(* IEC 61131-3 sources: beckhoffAutomationInterface/ST/Shark/App/Shark/FunctionBlocks, 11 files *)

(* ---- FB_ChillerManager.st ---- *)
(*
FB_ChillerManager — Controls chiller power and water valves.
Migrated from old FB_ChillerManager. Uses I_DigitalOutput from DO subsystem.
3 outputs: ChillerPower, ChuckWaterIn valve, ChuckWaterOut valve.
*)
FUNCTION_BLOCK FB_ChillerManager
VAR
    _ipChillerPower   : I_DigitalOutput;
    _ipWaterInValve   : I_DigitalOutput;
    _ipWaterOutValve  : I_DigitalOutput;
    _bInitialized     : BOOL := FALSE;
END_VAR

METHOD PUBLIC Init : BOOL
VAR_INPUT
    ipChillerPower  : I_DigitalOutput;
    ipWaterInValve  : I_DigitalOutput;
    ipWaterOutValve : I_DigitalOutput;
END_VAR
    IF ipChillerPower = 0 OR ipWaterInValve = 0 OR ipWaterOutValve = 0 THEN
        GVL_ErrorLogger.Logger.LogError(
            sSource  := 'ChillerManager.Init',
            eErrorId := E_ErrorId.ERR_GEN_NULL_POINTER,
            sContext := 'null interface pointer'
        );
        RETURN;
    END_IF
    _ipChillerPower := ipChillerPower;
    _ipWaterInValve := ipWaterInValve;
    _ipWaterOutValve := ipWaterOutValve;
    _bInitialized := TRUE;
    Init := TRUE;
END_METHOD

METHOD PUBLIC SetChillerPower
VAR_INPUT
    bOn : BOOL;
END_VAR
    _SetOutput(ipOutput := _ipChillerPower, bValue := bOn);
END_METHOD

METHOD PUBLIC SetWaterInValve
VAR_INPUT
    bOpen : BOOL;
END_VAR
    _SetOutput(ipOutput := _ipWaterInValve, bValue := bOpen);
END_METHOD

METHOD PUBLIC SetWaterOutValve
VAR_INPUT
    bOpen : BOOL;
END_VAR
    _SetOutput(ipOutput := _ipWaterOutValve, bValue := bOpen);
END_METHOD

METHOD PRIVATE _SetOutput
VAR_INPUT
    ipOutput : I_DigitalOutput;
    bValue   : BOOL;
END_VAR
    IF NOT _bInitialized THEN RETURN; END_IF
    ipOutput.SetOutput(bValue);
END_METHOD

PROPERTY PUBLIC IsChillerOn : BOOL
    GET
        IF _bInitialized AND_THEN _ipChillerPower <> 0 THEN
            IsChillerOn := _ipChillerPower.GetOutput();
        END_IF
    END_GET
END_PROPERTY

END_FUNCTION_BLOCK

(* ---- FB_ChuckVacuumSystem.st ---- *)
// Shark Chuck Vacuum System
//
// Shark hardware topology:
//   - Dedicated vacuum pump (PUMP_CHK_VAC) — toggled by this subsystem
//   - 2-way zone valves (VALV_CHK_LZ1/2/3) — open = vacuum applied
//   - Explicit vent valve (VALV_CHK_VENT) — must be closed before holding
//   - Single analog vacuum sensor (PSNS_CHK_VAC)
//
// Threshold semantics: rThreshold is in the same engineering units as the
// analog sensor; held when measurement < rThreshold, released when > rThreshold.
FUNCTION_BLOCK FB_ChuckVacuumSystem IMPLEMENTS I_ChuckVacuumSystem
VAR
    _bInitialized   : BOOL := FALSE;
    _bError         : BOOL := FALSE;

    _ipPump         : I_DigitalOutput;
    _ipValveLZ1     : I_Valve;
    _ipValveLZ2     : I_Valve;
    _ipValveLZ3     : I_Valve;
    _ipVentValve    : I_Valve;
    _ipVacuumSensor : I_Sensor;
END_VAR

VAR CONSTANT
    MAX_ZONES : INT := 3;
END_VAR

METHOD PUBLIC Init : BOOL
VAR_INPUT
    ipProvider : I_HardwareProvider;
END_VAR
    _bInitialized := FALSE;
    _bError := FALSE;

    IF ipProvider = 0 THEN
        GVL_ErrorLogger.Logger.LogError('FB_ChuckVacuumSystem', E_ErrorId.ERR_GEN_NULL_POINTER, 'Provider is null');
        RETURN;
    END_IF

    _ipPump := ipProvider.GetDigitalOutput(E_DigitalOutputIdentifier.PUMP_CHK_VAC);
    _ipValveLZ1 := ipProvider.GetValve(E_ValveIdentifier.VALV_CHK_LZ1);
    _ipValveLZ2 := ipProvider.GetValve(E_ValveIdentifier.VALV_CHK_LZ2);
    _ipValveLZ3 := ipProvider.GetValve(E_ValveIdentifier.VALV_CHK_LZ3);
    _ipVentValve := ipProvider.GetValve(E_ValveIdentifier.VALV_CHK_VENT);
    _ipVacuumSensor := ipProvider.GetPressureSensor(E_PressureSensorIdentifier.PSNS_CHK_VAC);

    IF _ipPump = 0 OR _ipValveLZ1 = 0 OR _ipVentValve = 0 OR _ipVacuumSensor = 0 THEN
        GVL_ErrorLogger.Logger.LogError('FB_ChuckVacuumSystem', E_ErrorId.ERR_GEN_NULL_POINTER, 'Required chuck vacuum hardware missing');
        RETURN;
    END_IF

    _bInitialized := TRUE;
    Init := TRUE;
END_METHOD

METHOD PUBLIC IsInitialized : BOOL
    IsInitialized := _bInitialized;
END_METHOD

METHOD PUBLIC IsError : BOOL
    IsError := _bError;
END_METHOD

METHOD PUBLIC GetMaxZoneCount : INT
    GetMaxZoneCount := MAX_ZONES;
END_METHOD

// Shark: close vent and ensure dedicated pump is on.
METHOD PUBLIC PrepareForHold : BOOL
    IF NOT _bInitialized THEN RETURN; END_IF
    _ipVentValve.Close();
    IF NOT _ipPump.GetOutput() THEN
        _ipPump.SetOutput(TRUE);
    END_IF
    PrepareForHold := TRUE;
END_METHOD

// Shark: open vent to atmosphere. Caller closes zones separately.
METHOD PUBLIC BeginRelease : BOOL
    IF NOT _bInitialized THEN RETURN; END_IF
    _ipVentValve.Open();
    BeginRelease := TRUE;
END_METHOD

// Shark: turn off dedicated chuck vacuum pump.
METHOD PUBLIC FinishRelease : BOOL
    IF NOT _bInitialized THEN RETURN; END_IF
    _ipPump.SetOutput(FALSE);
    FinishRelease := TRUE;
END_METHOD

METHOD PUBLIC OpenZone : BOOL
VAR_INPUT
    nZone : INT;
END_VAR
    OpenZone := _SetZoneState(nZone := nZone, bOpen := TRUE);
END_METHOD

METHOD PUBLIC CloseZone : BOOL
VAR_INPUT
    nZone : INT;
END_VAR
    CloseZone := _SetZoneState(nZone := nZone, bOpen := FALSE);
END_METHOD

// Analog sensor: vacuum held when pressure < threshold.
// nActiveZoneCount is ignored — single sensor measures shared vacuum manifold.
METHOD PUBLIC IsVacuumHeld : BOOL
VAR_INPUT
    nActiveZoneCount : INT;
    rThreshold       : LREAL;
END_VAR
    IF NOT _bInitialized THEN RETURN; END_IF
    IsVacuumHeld := (_ipVacuumSensor.GetMeasurement() < rThreshold);
END_METHOD

// Analog sensor: vacuum released when pressure > threshold.
METHOD PUBLIC IsVacuumReleased : BOOL
VAR_INPUT
    rThreshold : LREAL;
END_VAR
    IF NOT _bInitialized THEN RETURN; END_IF
    IsVacuumReleased := (_ipVacuumSensor.GetMeasurement() > rThreshold);
END_METHOD

METHOD PUBLIC Reset : BOOL
    _bError := FALSE;
    IF _ipValveLZ1 <> 0 AND_THEN _ipValveLZ1.IsError() THEN _ipValveLZ1.Reset(); END_IF
    IF _ipValveLZ2 <> 0 AND_THEN _ipValveLZ2.IsError() THEN _ipValveLZ2.Reset(); END_IF
    IF _ipValveLZ3 <> 0 AND_THEN _ipValveLZ3.IsError() THEN _ipValveLZ3.Reset(); END_IF
    IF _ipVentValve <> 0 AND_THEN _ipVentValve.IsError() THEN _ipVentValve.Reset(); END_IF
    Reset := TRUE;
END_METHOD

METHOD PRIVATE _SetZoneState : BOOL
VAR_INPUT
    nZone : INT;
    bOpen : BOOL;
END_VAR
    IF NOT _bInitialized THEN RETURN; END_IF

    CASE nZone OF
        1:
            IF _ipValveLZ1 = 0 THEN RETURN; END_IF
            IF bOpen THEN _ipValveLZ1.Open(); ELSE _ipValveLZ1.Close(); END_IF
        2:
            IF _ipValveLZ2 = 0 THEN RETURN; END_IF
            IF bOpen THEN _ipValveLZ2.Open(); ELSE _ipValveLZ2.Close(); END_IF
        3:
            IF _ipValveLZ3 = 0 THEN RETURN; END_IF
            IF bOpen THEN _ipValveLZ3.Open(); ELSE _ipValveLZ3.Close(); END_IF
        ELSE
            RETURN;
    END_CASE

    _SetZoneState := TRUE;
END_METHOD

END_FUNCTION_BLOCK

(* ---- FB_CommandReceiver.st ---- *)
(*
FB_CommandReceiver — Receives JSON commands from ADS byte stream and dispatches
to hardware provider, spectrometer, and sequence engine.

ADS Pattern:
  DALP Manager (.NET) writes JSON as raw bytes into AdsStream[0..4095].
  This FB polls every scan: if non-zero → parse JSON → dispatch → clear buffer.

Debug:
  Each command has a corresponding stDbgXxx struct and bDbgTrigXxx BOOL.
  Set struct fields and trigger from TwinCAT online to execute any command
  through the same code path as the Pilot.

Handles all command types from E_Command:
  Subsystem:    SetValve, SetMFCFlowRate, SetPressureController, SetHeaterZone,
                SetSwitch, ErrorAcknowledge
  Sequence:     SetTemperatureGradients, CancelProcess, StartBubblerFlow,
                StopBubblerFlow, StartPurge, HoldReleaseSample,
                StartSpotDeposition, StartBubblerLeakTest
  Spectrometer: SetSpectrometerData, SetSpectrometerDark

Requires Tc3_JsonXml library for FB_JsonDomParser + FB_JsonReadWriteDataType.
*)
FUNCTION_BLOCK FB_CommandReceiver
VAR
    AdsStream              : ARRAY[0..4095] OF BYTE;
    ZeroArray              : ARRAY[0..4095] OF BYTE;
    sCommand               : STRING(4096);
    sLastCommandParsed     : STRING(4096);
    SuccessCommandCount    : UDINT := 0;
    ErrorCommandCount      : UDINT := 0;

    fbJson                 : FB_JsonDomParser;
    jsonDoc                : Tc3_JsonXml.PVOID;
    jsonProp               : SJsonValue;
    fbJsonDataType         : FB_JsonReadWriteDataType;

    _nCommand              : DINT;
    _nCommandIndex         : DINT;

    _ipHardware            : I_HardwareProvider;
    _ipSpectrometer        : I_Spectrometer;
    _refOrchestrator       : REFERENCE TO FB_SequenceOrchestrator;
    _rTempDisableThreshold : REAL := 0.0;   // degC if any zone's setpoint is below this, disable all commands that could heat
    _bInitialized          : BOOL := FALSE;

    // Debug: set struct fields + trigger from TwinCAT online to test any command
    // Subsystem
    stDbgSetValve              : ST_CmdSetValve;
    bDbgTrigSetValve           : BOOL;
    stDbgSetFlowRate           : ST_CmdSetFlowRate;
    bDbgTrigSetFlowRate        : BOOL;
    stDbgSetPressure           : ST_CmdSetPressure;
    bDbgTrigSetPressure        : BOOL;
    stDbgSetHeatZone           : ST_CmdSetHeatZone;
    bDbgTrigSetHeatZone        : BOOL;
    stDbgSetSwitch             : ST_CmdSetSwitch;
    bDbgTrigSetSwitch          : BOOL;
    bDbgTrigErrorAck           : BOOL;
    // Sequence
    stDbgTempGradient          : ST_CmdSetTemperatureGradient;
    bDbgTrigTempGradient       : BOOL;
    bDbgTrigCancelProcess      : BOOL;
    stDbgBubblerFlow           : ST_CmdStartBubblerFlow;
    bDbgTrigBubblerFlow        : BOOL;
    stDbgStopBubblerFlow       : ST_CmdStopBubblerFlow;
    bDbgTrigStopBubblerFlow    : BOOL;
    stDbgPurge                 : ST_CmdPurge;
    bDbgTrigPurge              : BOOL;
    stDbgChuckZone             : ST_CmdSetChuckZone;
    bDbgTrigChuckZone          : BOOL;
    stDbgSpotDeposition        : ST_CmdSpotDeposition;
    bDbgTrigSpotDeposition     : BOOL;
    stDbgLeakTest              : ST_CmdBubblerLeakTest;
    bDbgTrigLeakTest           : BOOL;
    // Spectrometer
    stDbgSpectrometerData      : ST_DeviceSettings;
    bDbgTrigSpectrometerData   : BOOL;
    bDbgTrigSpectrometerDark   : BOOL;
END_VAR
VAR_OUTPUT
    nLastCommandIndex      : DINT;
END_VAR
VAR CONSTANT
    JSON_KEY_COMMAND             : STRING := 'command';
    JSON_KEY_INDEX               : STRING := 'index';
    JSON_KEY_PARAMETERS          : STRING := 'parameters';
    JSON_PARAM_BUFFER_SIZE       : UDINT  := 2048;
    // Minimum flow rate above which the inert gas inlet valve is opened.
    // At or below this threshold the valve is closed.
    INERT_FLOW_VALVE_THRESHOLD   : REAL   := 0.001;
END_VAR

    IF NOT _bInitialized THEN
        RETURN;
    END_IF

    IF MEMCMP(ADR(AdsStream), ADR(ZeroArray), SIZEOF(AdsStream)) <> 0 THEN
        sCommand := _ByteArrToString(ADR(AdsStream), SIZEOF(AdsStream));
        IF _ParseAndDispatch() THEN
            SuccessCommandCount := SuccessCommandCount + 1;
        ELSE
            ErrorCommandCount := ErrorCommandCount + 1;
        END_IF
        MEMSET(ADR(AdsStream), 0, SIZEOF(AdsStream));
        sLastCommandParsed := sCommand;
    END_IF

    // Debug triggers (set params + trigger from TwinCAT online)
    _ProcessDebugTriggers();

METHOD PUBLIC Init : BOOL
VAR_INPUT
    ipHardware     : I_HardwareProvider;
    ipSpectrometer : I_Spectrometer;
    rTempDisableThreshold : REAL;
    refOrchestrator : REFERENCE TO FB_SequenceOrchestrator;
END_VAR
    IF ipHardware = 0 OR ipSpectrometer = 0 THEN
        GVL_ErrorLogger.Logger.LogError(
            sSource  := 'CommandReceiver.Init',
            eErrorId := E_ErrorId.ERR_GEN_NULL_POINTER,
            sContext := 'invalid interface'
        );
        RETURN;
    END_IF
    IF NOT __ISVALIDREF(refOrchestrator) THEN
        GVL_ErrorLogger.Logger.LogError(
            sSource  := 'CommandReceiver.Init',
            eErrorId := E_ErrorId.ERR_GEN_NULL_POINTER,
            sContext := 'invalid orchestrator reference'
        );
        RETURN;
    END_IF
    _ipHardware            := ipHardware;
    _ipSpectrometer        := ipSpectrometer;
    _rTempDisableThreshold := rTempDisableThreshold;
    _refOrchestrator       REF= refOrchestrator;
    _bInitialized          := TRUE;
    Init := TRUE;
END_METHOD

METHOD PRIVATE _ParseAndDispatch : BOOL
VAR
    nError         : INT := 0;
    stSetValve     : ST_CmdSetValve;
    stSetFlowRate  : ST_CmdSetFlowRate;
    stSetPressure  : ST_CmdSetPressure;
    stSetHeatZone  : ST_CmdSetHeatZone;
    stSetHeatChannel : ST_CmdSetHeatChannel;
    stSetSwitch    : ST_CmdSetSwitch;
    stTempGrad     : ST_CmdSetTemperatureGradient;
    stBubblerFlow  : ST_CmdStartBubblerFlow;
    stStopBubbler  : ST_CmdStopBubblerFlow;
    stPurge        : ST_CmdPurge;
    stChuckZone    : ST_CmdSetChuckZone;
    stSpotDep      : ST_CmdSpotDeposition;
    stLeakTest     : ST_CmdBubblerLeakTest;
    stSpecData     : ST_DeviceSettings;
    eCmd           : E_Command;
END_VAR
    jsonDoc := fbJson.ParseDocument(sCommand);

    jsonProp := fbJson.FindMember(jsonDoc, JSON_KEY_COMMAND);
    IF jsonProp <> 0 THEN
        _nCommand := fbJson.GetInt(jsonProp);
    ELSE
        GVL_ErrorLogger.Logger.LogError(
            sSource   := 'CommandReceiver',
            eErrorId  := E_ErrorId.ERR_GEN_INVALID_PARAM,
            sContext  := 'missing command field in JSON',
            eSeverity := E_TcEventSeverity.Warning
        );
        _ParseAndDispatch := FALSE;
        RETURN;
    END_IF

    jsonProp := fbJson.FindMember(jsonDoc, JSON_KEY_INDEX);
    IF jsonProp <> 0 THEN
        _nCommandIndex := fbJson.GetInt(jsonProp);
    END_IF

    eCmd := DINT_TO_INT(_nCommand);
    CASE eCmd OF
        E_Command.SetValve:
            IF _ParseJsonParams('ST_CmdSetValve', SIZEOF(stSetValve), ADR(stSetValve)) THEN
                nError := _CmdSetValve(stCmd := stSetValve);
            ELSE nError := -1; END_IF
        E_Command.SetMFCFlowRate:
            IF _ParseJsonParams('ST_CmdSetFlowRate', SIZEOF(stSetFlowRate), ADR(stSetFlowRate)) THEN
                nError := _CmdSetMFCFlowRate(stCmd := stSetFlowRate);
            ELSE nError := -1; END_IF
        E_Command.SetPressureController:
            IF _ParseJsonParams('ST_CmdSetPressure', SIZEOF(stSetPressure), ADR(stSetPressure)) THEN
                nError := _CmdSetPressure(stCmd := stSetPressure);
            ELSE nError := -1; END_IF
        E_Command.SetHeaterZone:
            IF _ParseJsonParams('ST_CmdSetHeatZone', SIZEOF(stSetHeatZone), ADR(stSetHeatZone)) THEN
                nError := _CmdSetHeatZone(stCmd := stSetHeatZone);
            ELSE nError := -1; END_IF
        E_Command.SetHeaterChannel:
            IF _ParseJsonParams('ST_CmdSetHeatChannel', SIZEOF(stSetHeatChannel), ADR(stSetHeatChannel)) THEN
                nError := _CmdSetHeatChannel(stCmd := stSetHeatChannel);
            ELSE nError := -1; END_IF
        E_Command.SetSwitch:
            IF _ParseJsonParams('ST_CmdSetSwitch', SIZEOF(stSetSwitch), ADR(stSetSwitch)) THEN
                nError := _CmdSetSwitch(stCmd := stSetSwitch);
            ELSE nError := -1; END_IF
        E_Command.ErrorAcknowledge:
            nError := _CmdErrorAcknowledge();
        E_Command.SetTemperatureGradients:
            IF _ParseJsonParams('ST_CmdSetTemperatureGradient', SIZEOF(stTempGrad), ADR(stTempGrad)) THEN
                nError := _CmdSetTemperatureGradient(stCmd := stTempGrad);
            ELSE nError := -1; END_IF
        E_Command.CancelProcess:
            nError := _CmdCancelProcess();
        E_Command.StartBubblerFlow:
            IF _ParseJsonParams('ST_CmdStartBubblerFlow', SIZEOF(stBubblerFlow), ADR(stBubblerFlow)) THEN
                nError := _CmdStartBubblerFlow(stCmd := stBubblerFlow);
            ELSE nError := -1; END_IF
        E_Command.StopBubblerFlow:
            IF _ParseJsonParams('ST_CmdStopBubblerFlow', SIZEOF(stStopBubbler), ADR(stStopBubbler)) THEN
                nError := _CmdStopBubblerFlow(stCmd := stStopBubbler);
            ELSE nError := -1; END_IF
        E_Command.StartPurge:
            IF _ParseJsonParams('ST_CmdPurge', SIZEOF(stPurge), ADR(stPurge)) THEN
                nError := _CmdStartPurge(stCmd := stPurge);
            ELSE nError := -1; END_IF
        E_Command.HoldReleaseSample:
            IF _ParseJsonParams('ST_CmdSetChuckZone', SIZEOF(stChuckZone), ADR(stChuckZone)) THEN
                nError := _CmdHoldReleaseSample(stCmd := stChuckZone);
            ELSE nError := -1; END_IF
        E_Command.StartSpotDeposition:
            IF _ParseJsonParams('ST_CmdSpotDeposition', SIZEOF(stSpotDep), ADR(stSpotDep)) THEN
                nError := _CmdStartSpotDeposition(stCmd := stSpotDep);
            ELSE nError := -1; END_IF
        E_Command.StartBubblerLeakTest:
            IF _ParseJsonParams('ST_CmdBubblerLeakTest', SIZEOF(stLeakTest), ADR(stLeakTest)) THEN
                nError := _CmdStartBubblerLeakTest(stCmd := stLeakTest);
            ELSE nError := -1; END_IF
        E_Command.SetSpectrometerData:
            IF _ParseJsonParams('ST_DeviceSettings', SIZEOF(stSpecData), ADR(stSpecData)) THEN
                nError := _CmdSetSpectrometerData(stSettings := stSpecData);
            ELSE nError := -1; END_IF
        E_Command.SetSpectrometerDark:
            nError := _CmdSetSpectrometerDark();
    ELSE
        GVL_ErrorLogger.Logger.LogError(
            sSource   := 'CommandReceiver',
            eErrorId  := E_ErrorId.ERR_GEN_INVALID_PARAM,
            sContext  := CONCAT('unknown command ', CONCAT(TO_STRING(eCmd), CONCAT(' (', CONCAT(DINT_TO_STRING(_nCommand), ')')))),
            eSeverity := E_TcEventSeverity.Warning
        );
        _ParseAndDispatch := FALSE;
        RETURN;
    END_CASE

    IF nError = 0 THEN
        nLastCommandIndex := _nCommandIndex;
        _ParseAndDispatch := TRUE;
    ELSE
        GVL_ErrorLogger.Logger.LogError(
            sSource   := 'CommandReceiver',
            eErrorId  := E_ErrorId.ERR_GEN_INTERNAL,
            sContext  := CONCAT('command failed ', CONCAT(TO_STRING(eCmd), CONCAT(' (', CONCAT(DINT_TO_STRING(_nCommand), ')')))),
            eSeverity := E_TcEventSeverity.Warning
        );
        _ParseAndDispatch := FALSE;
    END_IF
END_METHOD

METHOD PRIVATE _ParseJsonParams : BOOL
VAR_INPUT
    sTypeName : STRING;
    nSize     : UDINT;
    pDest     : PVOID;
END_VAR
VAR
    sParamJson : STRING(JSON_PARAM_BUFFER_SIZE);
    nLen       : UDINT;
END_VAR
    jsonProp := fbJson.FindMember(jsonDoc, JSON_KEY_PARAMETERS);
    IF jsonProp = 0 THEN
        // No 'parameters' wrapper — fall back to using the full JSON directly
        sParamJson := sCommand;
    ELSE
        nLen := fbJson.GetJsonLength(jsonProp);
        fbJson.CopyJson(jsonProp, sParamJson, nLen);
    END_IF

    IF NOT fbJsonDataType.SetSymbolFromJson(sParamJson, sTypeName, nSize, pDest) THEN
        GVL_ErrorLogger.Logger.LogError(
            sSource   := 'CommandReceiver',
            eErrorId  := E_ErrorId.ERR_GEN_INVALID_PARAM,
            sContext  := CONCAT('failed to parse ', sTypeName),
            eSeverity := E_TcEventSeverity.Warning
        );
        _ParseJsonParams := FALSE;
        RETURN;
    END_IF
    _ParseJsonParams := TRUE;
END_METHOD

// =============================================================================
// COMMAND HANDLERS — Pure execution, no JSON parsing
// =============================================================================

METHOD PRIVATE _CmdSetValve : INT
VAR_INPUT
    stCmd : ST_CmdSetValve;
END_VAR
VAR
    ipValve : I_Valve;
    eValve  : E_ValveIdentifier;
END_VAR
    eValve := stCmd.valveId;
    GVL_ErrorLogger.Logger.LogInfo(
        sSource  := 'CommandReceiver',
        sContext := CONCAT('SetValve(', CONCAT(DINT_TO_STRING(_nCommand), CONCAT('): ', CONCAT(TO_STRING(eValve), CONCAT('(', CONCAT(INT_TO_STRING(stCmd.valveId), CONCAT(') enabled=', BOOL_TO_STRING(stCmd.enabled))))))))
    );
    ipValve := _ipHardware.GetValve(stCmd.valveId);
    IF ipValve <> 0 THEN
        IF stCmd.enabled THEN
            ipValve.Open();
        ELSE
            ipValve.Close();
        END_IF
    ELSE
        _CmdSetValve := -1;
    END_IF
END_METHOD

METHOD PRIVATE _CmdSetMFCFlowRate : INT
VAR_INPUT
    stCmd : ST_CmdSetFlowRate;
END_VAR
VAR
    ipController : I_Controller;
    ipInertValve : I_Valve;
    eMFC         : E_MFCIdentifier;
END_VAR
    eMFC := stCmd.mfcId;
    GVL_ErrorLogger.Logger.LogInfo(
        sSource  := 'CommandReceiver',
        sContext := CONCAT('SetMFCFlowRate(', CONCAT(DINT_TO_STRING(_nCommand), CONCAT('): ', CONCAT(TO_STRING(eMFC), CONCAT('(', CONCAT(INT_TO_STRING(stCmd.mfcId), CONCAT(') flowRate=', REAL_TO_STRING(stCmd.flowRate))))))))
    );
    ipController := _ipHardware.GetFlowController(stCmd.mfcId);
    IF ipController <> 0 THEN
        ipController.SetSetpoint(stCmd.flowRate);
        // When the inert MFC (MFCT_IG_01) is commanded, also control its inlet valve.
        IF eMFC = E_MFCIdentifier.MFCT_IG_01 THEN
            ipInertValve := _ipHardware.GetInertGasValve();
            IF ipInertValve <> 0 THEN
                IF stCmd.flowRate > INERT_FLOW_VALVE_THRESHOLD THEN
                    ipInertValve.Open();
                ELSE
                    ipInertValve.Close();
                END_IF
            END_IF
        END_IF
    ELSE
        _CmdSetMFCFlowRate := -1;
    END_IF
END_METHOD

METHOD PRIVATE _CmdSetPressure : INT
VAR_INPUT
    stCmd : ST_CmdSetPressure;
END_VAR
VAR
    ipController : I_Controller;
    ePressure    : E_PressureController;
END_VAR
    ePressure := stCmd.psctrlId;
    GVL_ErrorLogger.Logger.LogInfo(
        sSource  := 'CommandReceiver',
        sContext := CONCAT('SetPressureController(', CONCAT(DINT_TO_STRING(_nCommand), CONCAT('): ', CONCAT(TO_STRING(ePressure), CONCAT('(', CONCAT(INT_TO_STRING(stCmd.psctrlId), CONCAT(') pressure=', REAL_TO_STRING(stCmd.pressure))))))))
    );
    ipController := _ipHardware.GetPressureControllerById(stCmd.psctrlId);
    IF ipController <> 0 THEN
        ipController.SetSetpoint(stCmd.pressure);
    ELSE
        _CmdSetPressure := -1;
    END_IF
END_METHOD

METHOD PRIVATE _CmdSetHeatZone : INT
VAR_INPUT
    stCmd : ST_CmdSetHeatZone;
END_VAR
VAR
    ipController : I_Controller;
    eLegacyZone  : E_HeatZones;   // per-channel id sent by the DALP/Pilot client (1..15)
    eZone        : E_HeatZone;    // internal controllable zone id (1..13)
END_VAR
    // The legacy DALP/Pilot client addresses heater CHANNELS via E_HeatZones
    // (1..15), but SetHeaterZone operates on ZONES via E_HeatZone (1..13).
    // Reject any id that is not a defined E_HeatZones member, then translate.
    eLegacyZone := stCmd.zoneId;
    IF NOT _LegacyChannelToZone(eLegacy := eLegacyZone, eZone => eZone) THEN
        GVL_ErrorLogger.Logger.LogError(
            sSource   := 'CommandReceiver.SetHeatZone',
            eErrorId  := E_ErrorId.ERR_GEN_INVALID_PARAM,
            sContext  := CONCAT('invalid zoneId ', INT_TO_STRING(stCmd.zoneId)),
            eSeverity := E_TcEventSeverity.Warning
        );
        _CmdSetHeatZone := -1;
        RETURN;
    END_IF

    GVL_ErrorLogger.Logger.LogInfo(
        sSource  := 'CommandReceiver',
        sContext := CONCAT('SetHeatZone(', CONCAT(DINT_TO_STRING(_nCommand), CONCAT('): ', CONCAT(TO_STRING(eLegacyZone), CONCAT(' -> ', CONCAT(TO_STRING(eZone), CONCAT(' temp=', REAL_TO_STRING(stCmd.temp))))))))
    );

    ipController := _ipHardware.GetTemperatureController(eZone);
    IF ipController <> 0 THEN
        IF stCmd.temp > _rTempDisableThreshold THEN
            ipController.SetSetpoint(stCmd.temp);
            ipController.Enable(TRUE);
        ELSE
            ipController.Enable(FALSE);
        END_IF
    ELSE
        _CmdSetHeatZone := -1;
    END_IF
END_METHOD

(* Translate the legacy per-CHANNEL id (E_HeatZones, 1..15 — what the DALP/Pilot
   client sends) into the internal controllable ZONE id (E_HeatZone, 1..13).
   The 11 single-channel zones map 1:1. The two 2-channel zones each have two
   legacy channel ids that both resolve to the single owning zone:
       HETR_EXH_01 / HETR_EXH_02 -> HETR_EXH
       HETR_CHK_01 / HETR_CHK_02 -> HETR_CHK
   Commanding either channel id therefore enables the whole zone (FB_HeatZone
   fans Enable() out to every channel it owns).
   Returns TRUE and sets eZone on success; returns FALSE (leaving eZone
   untouched) for any value that is not a defined E_HeatZones member, so the
   caller can fail the command instead of acting on a wrong zone. *)
METHOD PRIVATE _LegacyChannelToZone : BOOL
VAR_INPUT
    eLegacy : E_HeatZones;
END_VAR
VAR_OUTPUT
    eZone : E_HeatZone;
END_VAR
    _LegacyChannelToZone := TRUE;
    CASE eLegacy OF
        E_HeatZones.HETR_HEAD_01 : eZone := E_HeatZone.HETR_HEAD;
        E_HeatZones.HETR_A_STR_01: eZone := E_HeatZone.HETR_A_STR;
        E_HeatZones.HETR_A_CMB_01: eZone := E_HeatZone.HETR_A_CMB;
        E_HeatZones.HETR_A_B1_01 : eZone := E_HeatZone.HETR_A_B1;
        E_HeatZones.HETR_A_B2_01 : eZone := E_HeatZone.HETR_A_B2;
        E_HeatZones.HETR_A_B3_01 : eZone := E_HeatZone.HETR_A_B3;
        E_HeatZones.HETR_B_STR_01: eZone := E_HeatZone.HETR_B_STR;
        E_HeatZones.HETR_B_CMB_01: eZone := E_HeatZone.HETR_B_CMB;
        E_HeatZones.HETR_B_B1_01 : eZone := E_HeatZone.HETR_B_B1;
        E_HeatZones.HETR_B_B2_01 : eZone := E_HeatZone.HETR_B_B2;
        E_HeatZones.HETR_B_B3_01 : eZone := E_HeatZone.HETR_B_B3;
        E_HeatZones.HETR_EXH_01,
        E_HeatZones.HETR_EXH_02  : eZone := E_HeatZone.HETR_EXH;
        E_HeatZones.HETR_CHK_01,
        E_HeatZones.HETR_CHK_02  : eZone := E_HeatZone.HETR_CHK;
    ELSE
        // Unknown id — not a defined E_HeatZones member. Fail; do not guess.
        _LegacyChannelToZone := FALSE;
    END_CASE
END_METHOD

METHOD PRIVATE _CmdSetHeatChannel : INT
VAR_INPUT
    stCmd : ST_CmdSetHeatChannel;
END_VAR
VAR
    ipController : I_Controller;
    eChannel     : E_HeatChannel;
END_VAR
    eChannel := stCmd.channelId;
    GVL_ErrorLogger.Logger.LogInfo(
        sSource  := 'CommandReceiver',
        sContext := CONCAT('SetHeatChannel(', CONCAT(DINT_TO_STRING(_nCommand), CONCAT('): ', CONCAT(TO_STRING(eChannel), CONCAT('(', CONCAT(INT_TO_STRING(stCmd.channelId), CONCAT(') temp=', REAL_TO_STRING(stCmd.temp))))))))
    );
    ipController := _ipHardware.GetTemperatureChannel(stCmd.channelId);
    IF ipController <> 0 THEN
        IF stCmd.temp > _rTempDisableThreshold THEN
            ipController.SetSetpoint(stCmd.temp);
            ipController.Enable(TRUE);
        ELSE
            ipController.Enable(FALSE);
        END_IF
    ELSE
        _CmdSetHeatChannel := -1;
    END_IF
END_METHOD

METHOD PRIVATE _CmdSetSwitch : INT
VAR_INPUT
    stCmd : ST_CmdSetSwitch;
END_VAR
VAR
    ipOutput : I_DigitalOutput;
    eDIO     : E_DIOIdentifier;
    eOutput  : E_DigitalOutputIdentifier;
END_VAR
    // switchId is sent by DALP Manager as an E_DIOIdentifier value (telemetry index 1..25).
    // Translate to E_DigitalOutputIdentifier before addressing the hardware.
    eDIO := stCmd.switchId;
    GVL_ErrorLogger.Logger.LogInfo(
        sSource  := 'CommandReceiver',
        sContext := CONCAT('SetSwitch(', CONCAT(DINT_TO_STRING(_nCommand), CONCAT('): ', CONCAT(TO_STRING(eDIO), CONCAT('(', CONCAT(INT_TO_STRING(stCmd.switchId), CONCAT(') enabled=', BOOL_TO_STRING(stCmd.enabled))))))))
    );

    CASE eDIO OF
        E_DIOIdentifier.LGHT_CMR_SIDE : eOutput := E_DigitalOutputIdentifier.LGHT_CMR_SIDE;
        E_DIOIdentifier.LGHT_CMR_TOP  : eOutput := E_DigitalOutputIdentifier.LGHT_CMR_TOP;
        E_DIOIdentifier.CHIL_PWR      : eOutput := E_DigitalOutputIdentifier.CHIL_PWR;
        // LGHT_SGN_RED, LGHT_SGN_YEL, LGHT_SGN_GRN are owned by FB_SignalLightController — not manually settable.
        E_DIOIdentifier.LOCK_DOOR_FL  : eOutput := E_DigitalOutputIdentifier.LOCK_DOOR_FL;
        E_DIOIdentifier.LOCK_DOOR_FR  : eOutput := E_DigitalOutputIdentifier.LOCK_DOOR_FR;
        E_DIOIdentifier.PUMP_CHK_VAC  : eOutput := E_DigitalOutputIdentifier.PUMP_CHK_VAC;
        E_DIOIdentifier.VALV_CHK_LZ1  : eOutput := E_DigitalOutputIdentifier.VALV_CHK_LZ1;
        E_DIOIdentifier.VALV_CHK_LZ2  : eOutput := E_DigitalOutputIdentifier.VALV_CHK_LZ2;
        E_DIOIdentifier.VALV_CHK_LZ3  : eOutput := E_DigitalOutputIdentifier.VALV_CHK_LZ3;
        E_DIOIdentifier.VALV_CHK_VENT : eOutput := E_DigitalOutputIdentifier.VALV_CHK_VENT;
    ELSE
        // DIO indices 9-17 are digital inputs (PRXS_DOOR_*) — not writable outputs.
        // DIO indices 24-25 are safety inputs (SAFE_STO_ON, SAFE_OVERRIDE) — not writable.
        GVL_ErrorLogger.Logger.LogError(
            sSource   := 'CommandReceiver.SetSwitch',
            eErrorId  := E_ErrorId.ERR_GEN_INVALID_PARAM,
            sContext  := CONCAT('DIO index ', CONCAT(TO_STRING(eDIO), ' is not a writable digital output')),
            eSeverity := E_TcEventSeverity.Warning
        );
        _CmdSetSwitch := -1;
        RETURN;
    END_CASE

    ipOutput := _ipHardware.GetDigitalOutput(eOutput);
    IF ipOutput <> 0 THEN
        ipOutput.SetOutput(stCmd.enabled);
    ELSE
        _CmdSetSwitch := -1;
    END_IF
END_METHOD

METHOD PRIVATE _CmdSetTemperatureGradient : INT
VAR_INPUT
    stCmd : ST_CmdSetTemperatureGradient;
END_VAR
    GVL_ErrorLogger.Logger.LogInfo(
        sSource  := 'CommandReceiver',
        sContext := CONCAT('SetTemperatureGradients: mode=', CONCAT(INT_TO_STRING(stCmd.enableMode), CONCAT(' head=', REAL_TO_STRING(stCmd.headTemp))))
    );
    IF NOT _refOrchestrator.StartHeating(stParams := stCmd) THEN
        _CmdSetTemperatureGradient := -1;
    END_IF
END_METHOD

METHOD PRIVATE _CmdErrorAcknowledge : INT
    GVL_System.bGlobalEmergencyStop := FALSE;
    _refOrchestrator.ErrorAcknowledge();
    GVL_ErrorLogger.Logger.LogInfo(
        sSource  := 'CommandReceiver',
        sContext := 'ErrorAcknowledge received'
    );
END_METHOD

METHOD PRIVATE _CmdCancelProcess : INT
    GVL_ErrorLogger.Logger.LogInfo(
        sSource  := 'CommandReceiver',
        sContext := 'CancelProcess'
    );
    IF NOT _refOrchestrator.SystemStop() THEN
        _CmdCancelProcess := -1;
    END_IF
END_METHOD

METHOD PRIVATE _CmdStartBubblerFlow : INT
VAR_INPUT
    stCmd : ST_CmdStartBubblerFlow;
END_VAR
VAR
    eSide : E_GasSide;
END_VAR
    eSide := stCmd.side;
    GVL_ErrorLogger.Logger.LogInfo(
        sSource  := 'CommandReceiver',
        sContext := CONCAT('StartBubblerFlow(', CONCAT(DINT_TO_STRING(_nCommand), CONCAT('): side=', CONCAT(TO_STRING(eSide), CONCAT('(', CONCAT(INT_TO_STRING(stCmd.side), CONCAT(') flow=', CONCAT(REAL_TO_STRING(stCmd.flowRate), CONCAT(' bubbler=', INT_TO_STRING(stCmd.bubblerIndex))))))))))
    );
    IF NOT _refOrchestrator.StartBubblerFlow(stParams := stCmd) THEN
        _CmdStartBubblerFlow := -1;
    END_IF
END_METHOD

METHOD PRIVATE _CmdStopBubblerFlow : INT
VAR_INPUT
    stCmd : ST_CmdStopBubblerFlow;
END_VAR
VAR
    eSide : E_GasSide;
END_VAR
    eSide := stCmd.side;
    GVL_ErrorLogger.Logger.LogInfo(
        sSource  := 'CommandReceiver',
        sContext := CONCAT('StopBubblerFlow(', CONCAT(DINT_TO_STRING(_nCommand), CONCAT('): side=', CONCAT(TO_STRING(eSide), CONCAT('(', CONCAT(INT_TO_STRING(stCmd.side), ')'))))))
    );
    IF NOT _refOrchestrator.StopBubblerFlow(stParams := stCmd) THEN
        _CmdStopBubblerFlow := -1;
    END_IF
END_METHOD

METHOD PRIVATE _CmdStartPurge : INT
VAR_INPUT
    stCmd : ST_CmdPurge;
END_VAR
VAR
    eMode : E_PurgeMode;
    eSide : E_GasSide;
END_VAR
    eMode := stCmd.mode;
    eSide := stCmd.side;
    GVL_ErrorLogger.Logger.LogInfo(
        sSource  := 'CommandReceiver',
        sContext := CONCAT('StartPurge(', CONCAT(DINT_TO_STRING(_nCommand), CONCAT('): ', CONCAT(TO_STRING(eMode), CONCAT('(', CONCAT(INT_TO_STRING(stCmd.mode), CONCAT(') side=', CONCAT(TO_STRING(eSide), CONCAT('(', CONCAT(INT_TO_STRING(stCmd.side), CONCAT(') bubbler=', INT_TO_STRING(stCmd.bubbler))))))))))))
    );
    IF NOT _refOrchestrator.StartPurge(stParams := stCmd) THEN
        _CmdStartPurge := -1;
    END_IF
END_METHOD

METHOD PRIVATE _CmdHoldReleaseSample : INT
VAR_INPUT
    stCmd     : ST_CmdSetChuckZone;
END_VAR
VAR
    iZone     : INT;
    stHold    : ST_ChuckVacuumHold;
    stRelease : ST_ChuckVacuumRelease;
END_VAR
    GVL_ErrorLogger.Logger.LogInfo(
        sSource  := 'CommandReceiver',
        sContext := CONCAT('HoldReleaseSample: hold=', CONCAT(BOOL_TO_STRING(stCmd.holdSample), CONCAT(' waferSize=', INT_TO_STRING(stCmd.size))))
    );
    IF stCmd.size < GVL_ChuckVacuumSystem.CHUCK_ZONE_SMALL_MAX THEN
        iZone := 1;
    ELSIF stCmd.size < GVL_ChuckVacuumSystem.CHUCK_ZONE_MEDIUM_MAX THEN
        iZone := 2;
    ELSE
        iZone := 3;
    END_IF

    IF stCmd.holdSample THEN
        stHold.iSelectZone := iZone;
        stHold.fLockPressureThreshold := stCmd.fPressureThreshold;
        stHold.tPressureTimeout := DINT_TO_TIME(stCmd.tPressureTimeout);
        IF NOT _refOrchestrator.StartChuckVacuumHold(stParams := stHold) THEN
            _CmdHoldReleaseSample := -1;
        END_IF
    ELSE
        stRelease.fReleasePressureThreshold := stCmd.fPressureThreshold;
        stRelease.tPressureTimeout := DINT_TO_TIME(stCmd.tPressureTimeout);
        IF NOT _refOrchestrator.StartChuckVacuumRelease(stParams := stRelease) THEN
            _CmdHoldReleaseSample := -1;
        END_IF
    END_IF
END_METHOD

METHOD PRIVATE _CmdStartSpotDeposition : INT
VAR_INPUT
    stCmd : ST_CmdSpotDeposition;
END_VAR
    GVL_ErrorLogger.Logger.LogInfo(
        sSource  := 'CommandReceiver',
        sContext := CONCAT('StartSpotDeposition: cycles=', CONCAT(DINT_TO_STRING(stCmd.nDepositionCycles), CONCAT(' precFlow=', REAL_TO_STRING(stCmd.fPrecursorFlowRate))))
    );
    IF NOT _refOrchestrator.StartSpotDeposition(stParams := stCmd) THEN
        _CmdStartSpotDeposition := -1;
    END_IF
END_METHOD

METHOD PRIVATE _CmdStartBubblerLeakTest : INT
VAR_INPUT
    stCmd : ST_CmdBubblerLeakTest;
END_VAR
VAR
    eSide : E_GasSide;
END_VAR
    eSide := stCmd.side;
    GVL_ErrorLogger.Logger.LogInfo(
        sSource  := 'CommandReceiver',
        sContext := CONCAT('StartBubblerLeakTest(', CONCAT(DINT_TO_STRING(_nCommand), CONCAT('): side=', CONCAT(TO_STRING(eSide), CONCAT('(', CONCAT(INT_TO_STRING(stCmd.side), CONCAT(') bubbler=', DINT_TO_STRING(stCmd.bubblerIndex))))))))
    );
    IF NOT _refOrchestrator.StartBubblerLeakTest(stParams := stCmd) THEN
        _CmdStartBubblerLeakTest := -1;
    END_IF
END_METHOD

METHOD PRIVATE _CmdSetSpectrometerData : INT
VAR_INPUT
    stSettings : ST_DeviceSettings;
END_VAR
    GVL_ErrorLogger.Logger.LogInfo(
        sSource  := 'CommandReceiver',
        sContext := CONCAT('SetSpectrometerData: scanRate=', CONCAT(UDINT_TO_STRING(stSettings.ScanRate), CONCAT(' avg=', UDINT_TO_STRING(stSettings.SpectrumAverage))))
    );
    _ipSpectrometer.SetFrequency(stSettings.ScanRate);
    _ipSpectrometer.SetLightIntensity(
        TargetLight := stSettings.LightTargetPercentage,
        AutoAdjust  := stSettings.IntensityAutoAdjust
    );
    _ipSpectrometer.SetAverageSample(stSettings.SpectrumAverage);
    _ipSpectrometer.SetSpectrumLimits(
        nStartRatio  := stSettings.SpectrumStart,
        nStopRatio   := stSettings.SpectrumStop,
        nTotalPixels := INT_TO_UDINT(GVL_Spectrometer.SPECTROMETER_PIXEL_COUNT)
    );
    _ipSpectrometer.SetQualityTreshold(stSettings.QualityThresholdPercentage);
END_METHOD

METHOD PRIVATE _CmdSetSpectrometerDark : INT
    GVL_ErrorLogger.Logger.LogInfo(
        sSource  := 'CommandReceiver',
        sContext := 'SetSpectrometerDark'
    );
    _ipSpectrometer.CalibrateDark(bExecute := TRUE);
END_METHOD

// =============================================================================
// DEBUG TRIGGERS — TwinCAT online: set struct fields, set trigger BOOL
// =============================================================================

METHOD PRIVATE _ProcessDebugTriggers
    // Subsystem
    IF bDbgTrigSetValve THEN
        bDbgTrigSetValve := FALSE;
        _CmdSetValve(stCmd := stDbgSetValve);
    END_IF
    IF bDbgTrigSetFlowRate THEN
        bDbgTrigSetFlowRate := FALSE;
        _CmdSetMFCFlowRate(stCmd := stDbgSetFlowRate);
    END_IF
    IF bDbgTrigSetPressure THEN
        bDbgTrigSetPressure := FALSE;
        _CmdSetPressure(stCmd := stDbgSetPressure);
    END_IF
    IF bDbgTrigSetHeatZone THEN
        bDbgTrigSetHeatZone := FALSE;
        _CmdSetHeatZone(stCmd := stDbgSetHeatZone);
    END_IF
    IF bDbgTrigSetSwitch THEN
        bDbgTrigSetSwitch := FALSE;
        _CmdSetSwitch(stCmd := stDbgSetSwitch);
    END_IF
    IF bDbgTrigErrorAck THEN
        bDbgTrigErrorAck := FALSE;
        _CmdErrorAcknowledge();
    END_IF

    // Sequence
    IF bDbgTrigTempGradient THEN
        bDbgTrigTempGradient := FALSE;
        _CmdSetTemperatureGradient(stCmd := stDbgTempGradient);
    END_IF
    IF bDbgTrigCancelProcess THEN
        bDbgTrigCancelProcess := FALSE;
        _CmdCancelProcess();
    END_IF
    IF bDbgTrigBubblerFlow THEN
        bDbgTrigBubblerFlow := FALSE;
        _CmdStartBubblerFlow(stCmd := stDbgBubblerFlow);
    END_IF
    IF bDbgTrigStopBubblerFlow THEN
        bDbgTrigStopBubblerFlow := FALSE;
        _CmdStopBubblerFlow(stCmd := stDbgStopBubblerFlow);
    END_IF
    IF bDbgTrigPurge THEN
        bDbgTrigPurge := FALSE;
        _CmdStartPurge(stCmd := stDbgPurge);
    END_IF
    IF bDbgTrigChuckZone THEN
        bDbgTrigChuckZone := FALSE;
        _CmdHoldReleaseSample(stCmd := stDbgChuckZone);
    END_IF
    IF bDbgTrigSpotDeposition THEN
        bDbgTrigSpotDeposition := FALSE;
        _CmdStartSpotDeposition(stCmd := stDbgSpotDeposition);
    END_IF
    IF bDbgTrigLeakTest THEN
        bDbgTrigLeakTest := FALSE;
        _CmdStartBubblerLeakTest(stCmd := stDbgLeakTest);
    END_IF

    // Spectrometer
    IF bDbgTrigSpectrometerData THEN
        bDbgTrigSpectrometerData := FALSE;
        _CmdSetSpectrometerData(stSettings := stDbgSpectrometerData);
    END_IF
    IF bDbgTrigSpectrometerDark THEN
        bDbgTrigSpectrometerDark := FALSE;
        _CmdSetSpectrometerDark();
    END_IF
END_METHOD

METHOD PRIVATE _ByteArrToString : STRING(4096)
VAR_INPUT
    pbyBuf : POINTER TO BYTE;
    diLen  : DINT;
END_VAR
VAR
    sResult  : STRING(4096) := '';
    nCopyLen : DINT;
END_VAR
    nCopyLen := MIN(diLen, 4095);
    MEMCPY(ADR(sResult), pbyBuf, TO_UDINT(nCopyLen));
    _ByteArrToString := sResult;
END_METHOD

END_FUNCTION_BLOCK

(* ---- FB_DALP.st ---- *)
(*
FB_DALP — Legacy client compatibility wrapper.

Exposes the exact ADS symbol contract the old C# DALP Manager expects:
  * MAIN.fbDALP.stTelemetry  (ST_Atlant3d_Telemetry, alias of ST_MachineTelemetry)
  * MAIN.fbDALP.AdsStream    (ARRAY[0..4095] OF BYTE, command write path)

This FB does not own any subsystem logic. It is a thin pass-through:
  1. Each scan, copy the new publisher's stTelemetry into our own
     stTelemetry (struct types alias each other, so the assignment is
     byte-for-byte equivalent).
  2. Overwrite the HETR_ array per-CHANNEL (not per-zone) so the legacy
     client's E_HeatZones iteration (15 entries) gets the right data.
  3. Forward any bytes the client wrote into AdsStream to the receiver's
     buffer, then clear the local buffer.

DELETE THIS FOLDER ONCE THE CLIENT IS UPDATED. See README.md.
*)
FUNCTION_BLOCK FB_DALP
VAR
    stTelemetry       : ST_Atlant3d_Telemetry;
    AdsStream         : ARRAY[0..4095] OF BYTE;
    _ZeroArray        : ARRAY[0..4095] OF BYTE;

    _refPublisher     : REFERENCE TO FB_TelemetryPublisher;
    _refReceiver      : REFERENCE TO FB_CommandReceiver;
    _refTempSub       : REFERENCE TO FB_TemperatureSubsystem;

    _bInitialized     : BOOL := FALSE;
END_VAR

    IF NOT _bInitialized THEN
        RETURN;
    END_IF

    // 1. Mirror the new publisher's full telemetry (identical struct shape via alias)
    stTelemetry := _refPublisher.stTelemetry;

    // 2. Re-fill HETR_ per-CHANNEL for the legacy client (15 entries on Shark)
    _UpdateHeatersPerChannel();

    // 3. Forward any client-written command bytes to the receiver
    IF MEMCMP(ADR(AdsStream), ADR(_ZeroArray), SIZEOF(AdsStream)) <> 0 THEN
        MEMCPY(
            destAddr := ADR(_refReceiver.AdsStream),
            srcAddr  := ADR(AdsStream),
            n        := SIZEOF(AdsStream)
        );
        MEMSET(ADR(AdsStream), 0, SIZEOF(AdsStream));
    END_IF

METHOD PUBLIC Init : BOOL
VAR_INPUT
    refPublisher : REFERENCE TO FB_TelemetryPublisher;
    refReceiver  : REFERENCE TO FB_CommandReceiver;
    refTempSub   : REFERENCE TO FB_TemperatureSubsystem;
END_VAR
    IF NOT __ISVALIDREF(refPublisher) THEN RETURN; END_IF
    IF NOT __ISVALIDREF(refReceiver)  THEN RETURN; END_IF
    IF NOT __ISVALIDREF(refTempSub)   THEN RETURN; END_IF

    _refPublisher REF= refPublisher;
    _refReceiver  REF= refReceiver;
    _refTempSub   REF= refTempSub;
    _bInitialized := TRUE;
    Init := TRUE;
END_METHOD

(* Per-CHANNEL heater telemetry for the legacy client.
   Iterates every (zone, channel) pair and writes HETR_[globalIdx]. *)
{attribute 'estimated-stack-usage' := '500'}
METHOD PRIVATE _UpdateHeatersPerChannel
VAR
    iZone       : INT;
    c           : INT;
    nCount      : INT;
    nGlobalIdx  : INT;
    ipChannel   : I_Controller;
    stCtrl      : ST_ControllerStatus;
END_VAR
    FOR iZone := 1 TO GVL_TemperatureZones.CONTROLLABLE_ZONE_MAX DO
        nCount := GVL_TemperatureZoneConfig.ZONE_CONFIG[iZone].nChannelCount;
        FOR c := 1 TO nCount DO
            nGlobalIdx := _refTempSub.GetChannelGlobalIndex(eZone := iZone, nChannelIdx := c);
            IF nGlobalIdx < 1 THEN CONTINUE; END_IF

            ipChannel := _refTempSub.GetChannel(eZone := iZone, nChannelIdx := c);
            IF ipChannel = 0 THEN CONTINUE; END_IF

            stCtrl := ipChannel.GetStatus();
            stTelemetry.HETR_[nGlobalIdx].Enable             := stCtrl.bEnabled;
            stTelemetry.HETR_[nGlobalIdx].TempAvg            := TO_REAL(stCtrl.rMeasuredValue);
            stTelemetry.HETR_[nGlobalIdx].SP                 := TO_REAL(stCtrl.rSetpoint);
            stTelemetry.HETR_[nGlobalIdx].TemperatureReached := stCtrl.bAtSetpoint;
            stTelemetry.HETR_[nGlobalIdx].Status             := SEL(
                stCtrl.stError.eErrorId = E_ErrorId.NO_ERROR, INT#1, INT#0);
        END_FOR
    END_FOR
END_METHOD

END_FUNCTION_BLOCK

(* ---- FB_DoorsManager.st ---- *)
(*
FB_DoorsManager — Shark-specific door wiring. Implements I_DoorSystem (Facade).

Facade pattern: presents the I_DoorSystem surface to sequence and safety code;
hides the lock/sensor graph and all Shark identifier knowledge from callers.

Layout: 9 proximity sensors, 2 door locks.
  Lock 1 FL (Front Left)  → sensors PRXS_DOOR_LT, PRXS_DOOR_LM
  Lock 2 FR (Front Right) → sensors PRXS_DOOR_RT, PRXS_DOOR_RM
  Remaining sensors (LB, RB, BML, BMR, BMB) are standalone monitoring only.

Sensor index assumption: E_DigitalInputIdentifier door enum values are dense
and align 1:1 with _afbSensors[1..SENSOR_COUNT]. If the enum is renumbered
this mapping must be revisited.
*)
FUNCTION_BLOCK FB_DoorsManager IMPLEMENTS I_DoorSystem
VAR
    _afbSensors   : ARRAY[1..GVL_DoorSystem.DOOR_SENSOR_COUNT] OF FB_DoorSensor;
    _afbLocks     : ARRAY[1..GVL_DoorSystem.DOOR_LOCK_COUNT] OF FB_DoorLock;
    _bInitialized : BOOL := FALSE;
END_VAR

METHOD PUBLIC Init : BOOL
VAR_INPUT
    ipDISub : I_DigitalInputSubsystem;
    ipDOSub : I_DigitalOutputSubsystem;
END_VAR
VAR
    i : INT;
END_VAR
    IF ipDISub = 0 OR ipDOSub = 0 THEN
        GVL_ErrorLogger.Logger.LogError(
            sSource  := 'DoorsManager.Init',
            eErrorId := E_ErrorId.ERR_GEN_NULL_POINTER,
            sContext := 'invalid subsystem interface pointer'
        );
        RETURN;
    END_IF

    // Initialise all 9 standalone monitoring sensors.
    // Relies on dense enum alignment: sensor identifier i maps to _afbSensors[i].
    FOR i := 1 TO GVL_DoorSystem.DOOR_SENSOR_COUNT DO
        _afbSensors[i].Init(ipInput := ipDISub.GetInputByIndex(nInput := i));
    END_FOR

    // Lock 1 — Front Left
    _afbLocks[1].Init(
        ipOutput := ipDOSub.GetOutputByIndex(nOutput := E_DigitalOutputIdentifier.LOCK_DOOR_FL)
    );
    _afbLocks[1].AddSensor(ipInput := ipDISub.GetInputByIndex(nInput := E_DigitalInputIdentifier.PRXS_DOOR_LT));
    _afbLocks[1].AddSensor(ipInput := ipDISub.GetInputByIndex(nInput := E_DigitalInputIdentifier.PRXS_DOOR_LM));

    // Lock 2 — Front Right
    _afbLocks[2].Init(
        ipOutput := ipDOSub.GetOutputByIndex(nOutput := E_DigitalOutputIdentifier.LOCK_DOOR_FR)
    );
    _afbLocks[2].AddSensor(ipInput := ipDISub.GetInputByIndex(nInput := E_DigitalInputIdentifier.PRXS_DOOR_RT));
    _afbLocks[2].AddSensor(ipInput := ipDISub.GetInputByIndex(nInput := E_DigitalInputIdentifier.PRXS_DOOR_RM));

    _bInitialized := TRUE;
    Init := TRUE;
END_METHOD

METHOD PUBLIC IsDoorClosed : BOOL
VAR_INPUT
    nSensorIndex : INT;
END_VAR
    IF nSensorIndex >= 1 AND nSensorIndex <= GVL_DoorSystem.DOOR_SENSOR_COUNT THEN
        IsDoorClosed := _afbSensors[nSensorIndex].IsClosed;
    END_IF
END_METHOD

METHOD PUBLIC IsLockActivated : BOOL
VAR_INPUT
    nLockIndex : INT;
END_VAR
    IF nLockIndex >= 1 AND nLockIndex <= GVL_DoorSystem.DOOR_LOCK_COUNT THEN
        IsLockActivated := _afbLocks[nLockIndex].IsLocked;
    END_IF
END_METHOD

METHOD PUBLIC LockDoor
VAR_INPUT
    nLockIndex : INT;
END_VAR
    IF nLockIndex >= 1 AND nLockIndex <= GVL_DoorSystem.DOOR_LOCK_COUNT THEN
        _afbLocks[nLockIndex].Lock();
    END_IF
END_METHOD

METHOD PUBLIC UnlockDoor
VAR_INPUT
    nLockIndex : INT;
END_VAR
    IF nLockIndex >= 1 AND nLockIndex <= GVL_DoorSystem.DOOR_LOCK_COUNT THEN
        _afbLocks[nLockIndex].Unlock();
    END_IF
END_METHOD

METHOD PUBLIC AreAllDoorsClosed : BOOL
VAR
    i : INT;
END_VAR
    AreAllDoorsClosed := TRUE;
    FOR i := 1 TO GVL_DoorSystem.DOOR_SENSOR_COUNT DO
        IF NOT _afbSensors[i].IsClosed THEN
            AreAllDoorsClosed := FALSE;
            RETURN;
        END_IF
    END_FOR
END_METHOD

END_FUNCTION_BLOCK

(* ---- FB_ExhaustController.st ---- *)
(*
FB_ExhaustController — Exhaust pump controller.

Keeps the exhaust pump energised at all times and optionally verifies
operation via an isolation valve and pressure sensor.

Configuration variants (set at Init time):
  A. Valve before sensor (bIsoValveBeforeSensor=TRUE, Shark):
       PUMP_ON → OPENING_VALVE → WAIT_PRESSURE → READY
  B. Sensor before valve, or no valve (bIsoValveBeforeSensor=FALSE):
       PUMP_ON → WAIT_PRESSURE → READY   (valve not managed here)
  C. Sensor only, no valve:
       PUMP_ON → WAIT_PRESSURE → READY
  D. Neither:
       PUMP_ON → READY

Pump output is re-driven every scan cycle — it cannot be silenced by
Halt() calls or any other external writer.
*)
FUNCTION_BLOCK FB_ExhaustController
VAR CONSTANT
    PRESSURE_THRESHOLD : LREAL := 0.4;   // bar — minimum to confirm pump health
    ISO_VALVE_OPEN_TIMEOUT  : TIME  := T#10S; // maximum wait for IsOpen() to return TRUE
    PRESSURE_BUILD_TIMEOUT  : TIME  := T#60S; // maximum wait for pressure to reach threshold
END_VAR
VAR
    _ipExhaustPump          : I_DigitalOutput;
    _ipIsoValve             : I_Valve;
    _ipPressureSensor       : I_Sensor;
    _bIsoValveBeforeSensor : BOOL;
    _eState                : E_ExhaustState := E_ExhaustState.INIT;
    _tonIsoValveOpen       : TON;
    _tonPressureBuild      : TON;
    _bInitialized           : BOOL := FALSE;
END_VAR

    IF NOT _bInitialized THEN
        RETURN;
    END_IF

    // Re-drive every scan — prevents any external SetOutput(FALSE) from lasting more than one cycle
    _ipExhaustPump.SetOutput(TRUE);

    CASE _eState OF

        E_ExhaustState.INIT:
            _eState := E_ExhaustState.PUMP_ON;

        E_ExhaustState.PUMP_ON:
            IF _ipIsoValve <> 0 AND_THEN _bIsoValveBeforeSensor THEN
                _eState := E_ExhaustState.OPENING_VALVE;
            ELSIF _ipPressureSensor <> 0 THEN
                _eState := E_ExhaustState.WAIT_PRESSURE;
            ELSE
                _eState := E_ExhaustState.READY;
            END_IF

        E_ExhaustState.OPENING_VALVE:
            _ipIsoValve.Open();
            _tonIsoValveOpen(IN := TRUE, PT := ISO_VALVE_OPEN_TIMEOUT);
            IF _ipIsoValve.IsOpen() THEN
                _tonIsoValveOpen(IN := FALSE);
                IF _ipPressureSensor <> 0 THEN
                    _eState := E_ExhaustState.WAIT_PRESSURE;
                ELSE
                    _eState := E_ExhaustState.READY;
                END_IF
            ELSIF _tonIsoValveOpen.Q THEN
                GVL_ErrorLogger.Logger.LogError(
                    sSource  := 'ExhaustController',
                    eErrorId := E_ErrorId.ERR_VALVE_FEEDBACK_TIMEOUT,
                    sContext := 'iso valve did not open within timeout',
                    fCurrentValue  := TO_REAL(TIME_TO_DWORD(_tonIsoValveOpen.ET)) / 1000.0,
                    fExpectedValue := TO_REAL(TIME_TO_DWORD(ISO_VALVE_OPEN_TIMEOUT)) / 1000.0,
                    sUnits := 's'
                );
                _eState := E_ExhaustState.ERROR;
            END_IF

        E_ExhaustState.WAIT_PRESSURE:
            _tonPressureBuild(IN := TRUE, PT := PRESSURE_BUILD_TIMEOUT);
            IF _ipPressureSensor.GetMeasurement() >= PRESSURE_THRESHOLD THEN
                _tonPressureBuild(IN := FALSE);
                _eState := E_ExhaustState.READY;
            ELSIF _tonPressureBuild.Q THEN
                GVL_ErrorLogger.Logger.LogError(
                    sSource  := 'ExhaustController',
                    eErrorId := E_ErrorId.ERR_GEN_TIMEOUT,
                    sContext := 'pressure threshold not reached',
                    fCurrentValue  := TO_REAL(_ipPressureSensor.GetMeasurement()),
                    fExpectedValue := TO_REAL(PRESSURE_THRESHOLD),
                    sUnits := 'bar'
                );
                _eState := E_ExhaustState.ERROR;
            END_IF

        E_ExhaustState.READY:
            ; // Pump always on — nothing to monitor

        E_ExhaustState.ERROR:
            ; // Stays here until Reset()

    END_CASE

METHOD PUBLIC Init : BOOL
VAR_INPUT
    ipExhaustPump          : I_DigitalOutput;
    ipIsoValve             : I_Valve  := 0;    // Optional — 0 if machine has no iso valve
    ipPressureSensor       : I_Sensor := 0;    // Optional — 0 if machine has no pressure sensor
    bIsoValveBeforeSensor  : BOOL     := FALSE; // TRUE = iso valve sits between pump and sensor (Shark);
                                                 // pressure is not meaningful until valve is open
END_VAR
    IF ipExhaustPump = 0 THEN
        GVL_ErrorLogger.Logger.LogError(
            sSource  := 'ExhaustController.Init',
            eErrorId := E_ErrorId.ERR_GEN_NULL_POINTER,
            sContext := 'null pump interface'
        );
        RETURN;
    END_IF
    _ipExhaustPump          := ipExhaustPump;
    _ipIsoValve             := ipIsoValve;
    _ipPressureSensor       := ipPressureSensor;
    _bIsoValveBeforeSensor  := bIsoValveBeforeSensor;
    _bInitialized           := TRUE;
    _eState                 := E_ExhaustState.INIT;
    Init := TRUE;
END_METHOD

METHOD PUBLIC Reset
    IF _bInitialized THEN
        _tonIsoValveOpen(IN := FALSE);
        _tonPressureBuild(IN := FALSE);
        IF _ipIsoValve <> 0 THEN
            _ipIsoValve.Close();
        END_IF
        _eState := E_ExhaustState.INIT;
    END_IF
END_METHOD

PROPERTY PUBLIC IsReady : BOOL
    GET
        IsReady := _eState = E_ExhaustState.READY;
    END_GET
END_PROPERTY

PROPERTY PUBLIC State : E_ExhaustState
    GET
        State := _eState;
    END_GET
END_PROPERTY

END_FUNCTION_BLOCK

(* ---- FB_HardwareProvider.st ---- *)
(* Hardware provider for Shark System (Dual-sided gas, Modbus pressure).
   Delegates Init and index-based subsystem access to FB_HardwareProviderBase.

   Shark-specific differences from PRO:
   - Per-side mix valves (VALV_A_MIX, VALV_B_MIX) instead of shared VALV_AB_MIX
   - Separate CM and HM vacuum isolation (DST_EXH vs CMB_EXH) instead of shared exhaust
   - Modbus pressure controllers via E_PressureController
    - 3 bubblers per side (no B-side gas-only lines)
    - No inert MFC side mapping (accessed via generic GetValve) *)
FUNCTION_BLOCK FB_HardwareProvider EXTENDS FB_HardwareProviderBase IMPLEMENTS I_HardwareProvider
VAR
    _nMaxBubblers : ARRAY[1..2] OF DINT := [3, 3];  // index matches E_GasSide: A_SIDE=1 → 3, B_SIDE=2 → 3
    _fbChuckVacuum         : FB_ChuckVacuumSystem;
    _bChuckVacuumInitTried : BOOL := FALSE;
END_VAR

// =============================================================================
// GENERIC GETTERS — thin wrappers delegating to base index-based helpers
// =============================================================================

METHOD GetValve : I_Valve
VAR_INPUT
    nIndex : INT;
END_VAR
    GetValve := SUPER^.GetValveByIndex(nIndex);
END_METHOD

METHOD GetDigitalOutput : I_DigitalOutput
VAR_INPUT
    nIndex : INT;
END_VAR
    GetDigitalOutput := SUPER^.GetOutputByIndex(nIndex);
END_METHOD

METHOD GetDigitalInput : I_DigitalInput
VAR_INPUT
    nIndex : INT;
END_VAR
    GetDigitalInput := SUPER^.GetInputByIndex(nIndex);
END_METHOD

METHOD GetPressureSensor : I_Sensor
VAR_INPUT
    nIndex : INT;
END_VAR
    GetPressureSensor := SUPER^.GetSensorByIndex(nIndex);
END_METHOD

METHOD GetFlowController : I_Controller
VAR_INPUT
    nIndex : INT;
END_VAR
    GetFlowController := SUPER^.GetFlowControllerByIndex(nIndex);
END_METHOD

METHOD GetPressureControllerById : I_Controller
VAR_INPUT
    nIndex : INT;
END_VAR
    GetPressureControllerById := SUPER^.GetPressureControllerByIndex(nIndex);
END_METHOD

METHOD GetTemperatureController : I_Controller
VAR_INPUT
    nIndex : INT;
END_VAR
    GetTemperatureController := SUPER^.GetTemperatureControllerByIndex(nIndex);
END_METHOD

METHOD GetTemperatureChannel : I_Controller
VAR_INPUT
    nGlobalIdx : INT;
END_VAR
    GetTemperatureChannel := SUPER^.GetTemperatureChannelByGlobalIndex(nGlobalIdx);
END_METHOD

// =============================================================================
// VALVE GETTERS - Side-abstracted
// =============================================================================

// Shark: One MFC valve per side (no extra gas lines)
METHOD GetGasIsoValve : I_Valve
VAR_INPUT
    eSide : E_GasSide;
    nBubblerIndex : DINT;
END_VAR
    IF eSide = E_GasSide.A_SIDE THEN
        GetGasIsoValve := GetValve(E_ValveIdentifier.VALV_A_MFC01);
    ELSE
        GetGasIsoValve := GetValve(E_ValveIdentifier.VALV_B_MFC01);
    END_IF
END_METHOD

// CM (Distributor) bubbler inlet valves
METHOD GetCMBubblerValve : I_Valve
VAR_INPUT
    eSide : E_GasSide;
    nBubblerIndex : DINT;
END_VAR
    nBubblerIndex := LIMIT(1, nBubblerIndex, 3);

    IF eSide = E_GasSide.A_SIDE THEN
        CASE nBubblerIndex OF
            1: GetCMBubblerValve := GetValve(E_ValveIdentifier.VALV_A_DST_B1);
            2: GetCMBubblerValve := GetValve(E_ValveIdentifier.VALV_A_DST_B2);
            3: GetCMBubblerValve := GetValve(E_ValveIdentifier.VALV_A_DST_B3);
        END_CASE
    ELSE
        CASE nBubblerIndex OF
            1: GetCMBubblerValve := GetValve(E_ValveIdentifier.VALV_B_DST_B1);
            2: GetCMBubblerValve := GetValve(E_ValveIdentifier.VALV_B_DST_B2);
            3: GetCMBubblerValve := GetValve(E_ValveIdentifier.VALV_B_DST_B3);
        END_CASE
    END_IF
END_METHOD

// HM (Combiner) bubbler outlet valves
METHOD GetHMBubblerValve : I_Valve
VAR_INPUT
    eSide : E_GasSide;
    nBubblerIndex : DINT;
END_VAR
    nBubblerIndex := LIMIT(1, nBubblerIndex, 3);

    IF eSide = E_GasSide.A_SIDE THEN
        CASE nBubblerIndex OF
            1: GetHMBubblerValve := GetValve(E_ValveIdentifier.VALV_A_CMB_B1);
            2: GetHMBubblerValve := GetValve(E_ValveIdentifier.VALV_A_CMB_B2);
            3: GetHMBubblerValve := GetValve(E_ValveIdentifier.VALV_A_CMB_B3);
        END_CASE
    ELSE
        CASE nBubblerIndex OF
            1: GetHMBubblerValve := GetValve(E_ValveIdentifier.VALV_B_CMB_B1);
            2: GetHMBubblerValve := GetValve(E_ValveIdentifier.VALV_B_CMB_B2);
            3: GetHMBubblerValve := GetValve(E_ValveIdentifier.VALV_B_CMB_B3);
        END_CASE
    END_IF
END_METHOD

METHOD GetCMPurgeValve : I_Valve
VAR_INPUT
    eSide : E_GasSide;
END_VAR
    IF eSide = E_GasSide.A_SIDE THEN
        GetCMPurgeValve := GetValve(E_ValveIdentifier.VALV_A_DST_PRG);
    ELSE
        GetCMPurgeValve := GetValve(E_ValveIdentifier.VALV_B_DST_PRG);
    END_IF
END_METHOD

METHOD GetHMPurgeValve : I_Valve
VAR_INPUT
    eSide : E_GasSide;
END_VAR
    IF eSide = E_GasSide.A_SIDE THEN
        GetHMPurgeValve := GetValve(E_ValveIdentifier.VALV_A_CMB_PRG);
    ELSE
        GetHMPurgeValve := GetValve(E_ValveIdentifier.VALV_B_CMB_PRG);
    END_IF
END_METHOD

// Shark: Separate CM and HM vacuum isolation (Distributor Exhaust vs Combiner Exhaust)
METHOD GetCMVacuumIsoValve : I_Valve
VAR_INPUT
    eSide : E_GasSide;
END_VAR
    IF eSide = E_GasSide.A_SIDE THEN
        GetCMVacuumIsoValve := GetValve(E_ValveIdentifier.VALV_A_DST_EXH);
    ELSE
        GetCMVacuumIsoValve := GetValve(E_ValveIdentifier.VALV_B_DST_EXH);
    END_IF
END_METHOD

METHOD GetHMVacuumIsoValve : I_Valve
VAR_INPUT
    eSide : E_GasSide;
END_VAR
    IF eSide = E_GasSide.A_SIDE THEN
        GetHMVacuumIsoValve := GetValve(E_ValveIdentifier.VALV_A_CMB_EXH);
    ELSE
        GetHMVacuumIsoValve := GetValve(E_ValveIdentifier.VALV_B_CMB_EXH);
    END_IF
END_METHOD

METHOD GetNozzleIsoValve : I_Valve
VAR_INPUT
    eSide : E_GasSide;
END_VAR
    IF eSide = E_GasSide.A_SIDE THEN
        GetNozzleIsoValve := GetValve(E_ValveIdentifier.VALV_A_STR);
    ELSE
        GetNozzleIsoValve := GetValve(E_ValveIdentifier.VALV_B_STR);
    END_IF
END_METHOD

// =============================================================================
// VALVE GETTERS - Common
// =============================================================================

// Shark has per-side mix valves (VALV_A_MIX, VALV_B_MIX), no shared mix valve.
// Returns 0 — use GetValve(E_ValveIdentifier.VALV_A_MIX) for direct access.
METHOD GetMixValve : I_Valve
    GetMixValve := 0;
END_METHOD

METHOD GetExhaustVacuumIsoValve : I_Valve
    GetExhaustVacuumIsoValve := GetValve(E_ValveIdentifier.VALV_EX_PUMP);
END_METHOD

// =============================================================================
// DIGITAL OUTPUT GETTERS
// =============================================================================

METHOD GetExhaustPump : I_DigitalOutput
    GetExhaustPump := GetDigitalOutput(E_DigitalOutputIdentifier.PUMP_AB_EXH);
END_METHOD

// =============================================================================
// SENSOR GETTERS - Side-abstracted
// =============================================================================

// CM (Distributor) pressure sensors
METHOD GetCMPressureSensor : I_Sensor
VAR_INPUT
    eSide : E_GasSide;
END_VAR
    IF eSide = E_GasSide.A_SIDE THEN
        GetCMPressureSensor := GetPressureSensor(E_PressureSensorIdentifier.PSNS_A_DST);
    ELSE
        GetCMPressureSensor := GetPressureSensor(E_PressureSensorIdentifier.PSNS_B_DST);
    END_IF
END_METHOD

// HM (Combiner/Hot Manifold) — Bronkhorst controller as sensor via __QUERYINTERFACE
METHOD GetHMPressureSensor : I_Sensor
VAR_INPUT
    eSide : E_GasSide;
END_VAR
    IF eSide = E_GasSide.A_SIDE THEN
        GetHMPressureSensor := SUPER^.GetPressureControllerAsSensor(E_PressureController.A_Side);
    ELSE
        GetHMPressureSensor := SUPER^.GetPressureControllerAsSensor(E_PressureController.B_Side);
    END_IF
END_METHOD

METHOD GetMFCFlowSensor : I_Sensor
VAR_INPUT
    eSide : E_GasSide;
END_VAR
    IF eSide = E_GasSide.A_SIDE THEN
        GetMFCFlowSensor := SUPER^.GetFlowControllerAsSensor(E_MFCIdentifier.MFCT_A_01);
    ELSE
        GetMFCFlowSensor := SUPER^.GetFlowControllerAsSensor(E_MFCIdentifier.MFCT_B_01);
    END_IF
END_METHOD

// =============================================================================
// SENSOR GETTERS - Common
// =============================================================================

METHOD GetExhaustPressureSensor : I_Sensor
    GetExhaustPressureSensor := GetPressureSensor(E_PressureSensorIdentifier.PSNS_AB_EXH);
END_METHOD

// =============================================================================
// CONTROLLER GETTERS - Side-abstracted
// =============================================================================

METHOD GetMFCController : I_Controller
VAR_INPUT
    eSide : E_GasSide;
END_VAR
    IF eSide = E_GasSide.A_SIDE THEN
        GetMFCController := SUPER^.GetFlowControllerByIndex(E_MFCIdentifier.MFCT_A_01);
    ELSE
        GetMFCController := SUPER^.GetFlowControllerByIndex(E_MFCIdentifier.MFCT_B_01);
    END_IF
END_METHOD

// Shark: Modbus Bronkhorst pressure controllers (E_PressureController)
METHOD GetPressureController : I_Controller
VAR_INPUT
    eSide : E_GasSide;
END_VAR
    IF eSide = E_GasSide.A_SIDE THEN
        GetPressureController := SUPER^.GetPressureControllerByIndex(E_PressureController.A_Side);
    ELSE
        GetPressureController := SUPER^.GetPressureControllerByIndex(E_PressureController.B_Side);
    END_IF
END_METHOD

// Inert Gas MFC Controller (Shark-only, used by SpotDeposition)
METHOD GetInertMFCController : I_Controller
    GetInertMFCController := SUPER^.GetFlowControllerByIndex(E_MFCIdentifier.MFCT_IG_01);
END_METHOD

// Inert Gas Valve (used by SpotDeposition)
METHOD GetInertGasValve : I_Valve
    GetInertGasValve := GetValve(E_ValveIdentifier.VALV_IG_MFC01);
END_METHOD

// Chuck Vacuum Subsystem — lazy-initialized on first request.
METHOD GetChuckVacuumSystem : I_ChuckVacuumSystem
    IF NOT _bChuckVacuumInitTried THEN
        _bChuckVacuumInitTried := TRUE;
        _fbChuckVacuum.Init(ipProvider := THIS^);
    END_IF
    GetChuckVacuumSystem := _fbChuckVacuum;
END_METHOD

// =============================================================================
// TEMPERATURE CONTROLLER GETTERS - Side-abstracted
// =============================================================================

METHOD GetHMTemperatureController : I_Controller
VAR_INPUT
    eSide : E_GasSide;
END_VAR
    IF eSide = E_GasSide.A_SIDE THEN
        GetHMTemperatureController := SUPER^.GetTemperatureControllerByIndex(E_HeatZone.HETR_A_CMB);
    ELSE
        GetHMTemperatureController := SUPER^.GetTemperatureControllerByIndex(E_HeatZone.HETR_B_CMB);
    END_IF
END_METHOD

METHOD GetUmbilicalTemperatureController : I_Controller
VAR_INPUT
    eSide : E_GasSide;
END_VAR
    IF eSide = E_GasSide.A_SIDE THEN
        GetUmbilicalTemperatureController := SUPER^.GetTemperatureControllerByIndex(E_HeatZone.HETR_A_STR);
    ELSE
        GetUmbilicalTemperatureController := SUPER^.GetTemperatureControllerByIndex(E_HeatZone.HETR_B_STR);
    END_IF
END_METHOD

METHOD GetBubblerTemperatureController : I_Controller
VAR_INPUT
    eSide : E_GasSide;
    nBubblerIndex : DINT;
END_VAR
    nBubblerIndex := LIMIT(1, nBubblerIndex, 3);

    IF eSide = E_GasSide.A_SIDE THEN
        CASE nBubblerIndex OF
            1: GetBubblerTemperatureController := SUPER^.GetTemperatureControllerByIndex(E_HeatZone.HETR_A_B1);
            2: GetBubblerTemperatureController := SUPER^.GetTemperatureControllerByIndex(E_HeatZone.HETR_A_B2);
            3: GetBubblerTemperatureController := SUPER^.GetTemperatureControllerByIndex(E_HeatZone.HETR_A_B3);
        END_CASE
    ELSE
        CASE nBubblerIndex OF
            1: GetBubblerTemperatureController := SUPER^.GetTemperatureControllerByIndex(E_HeatZone.HETR_B_B1);
            2: GetBubblerTemperatureController := SUPER^.GetTemperatureControllerByIndex(E_HeatZone.HETR_B_B2);
            3: GetBubblerTemperatureController := SUPER^.GetTemperatureControllerByIndex(E_HeatZone.HETR_B_B3);
        END_CASE
    END_IF
END_METHOD

// =============================================================================
// TEMPERATURE CONTROLLER GETTERS - Common
// =============================================================================

METHOD GetHeadTemperatureController : I_Controller
    GetHeadTemperatureController := SUPER^.GetTemperatureControllerByIndex(E_HeatZone.HETR_HEAD);
END_METHOD

METHOD GetExhaustTemperatureController : I_Controller
    GetExhaustTemperatureController := SUPER^.GetTemperatureControllerByIndex(E_HeatZone.HETR_EXH);
END_METHOD

METHOD GetChuckTemperatureController : I_Controller
    GetChuckTemperatureController := SUPER^.GetTemperatureControllerByIndex(E_HeatZone.HETR_CHK);
END_METHOD

// =============================================================================
// UTILITY & CONFIGURATION
// =============================================================================

// Shark has no gas-only lines — all bubblers are bubbler mode
METHOD IsGasMode : BOOL
VAR_INPUT
    eSide : E_GasSide;
    nBubblerIndex : DINT;
END_VAR
    IsGasMode := FALSE;
END_METHOD

METHOD GetMaxBubblerCount : DINT
VAR_INPUT
    eSide : E_GasSide;
END_VAR
    GetMaxBubblerCount := _nMaxBubblers[eSide];
END_METHOD

END_FUNCTION_BLOCK

(* ---- FB_SafetyManager.st ---- *)
(*
FB_SafetyManager — Safety state machine for Shark system.
*)
FUNCTION_BLOCK FB_SafetyManager IMPLEMENTS I_Errorable, I_SafetyStatus
VAR
    _eState              : E_SafetyState := E_SafetyState.ERROR;
    _nInitStep           : INT := 0;
    _bFirstCycle         : BOOL := TRUE;
    _bHeaterVoltagePresent : BOOL;

    // Edge triggers
    _rtNotSafe           : R_TRIG;
    _rtError             : R_TRIG;
    _rtVoltageOn         : R_TRIG;
    _ftVoltageOff        : F_TRIG;

    // Timers
    _tonSafetyStep       : TON;
    _tonStartupDelay     : TON;

    // Subsystem references (set via Init)
    _ipFlowSubsystem     : REFERENCE TO FB_FlowSubsystem;
    _bInitialized        : BOOL := FALSE;

    // Error surface (bridges TwinSAFE plane into the software error plane)
    _fbError             : FB_ErrorHandler;
END_VAR
VAR CONSTANT
    VOLTAGE_THRESHOLD    : REAL := 200.0;   // V — EL3443 heater voltage presence
    SAFETY_STEP_TIME     : TIME := T#100MS;
    STARTUP_DELAY        : TIME := T#5S;
END_VAR

IF NOT _bInitialized THEN
    RETURN;
END_IF

// --- Voltage monitoring ---
_bHeaterVoltagePresent := _CheckVoltage();
_rtVoltageOn(CLK := _bHeaterVoltagePresent);
_ftVoltageOff(CLK := _bHeaterVoltagePresent);

// --- Safety state machine ---
_tonSafetyStep.IN := TRUE;
_tonStartupDelay.IN := TRUE;
_tonStartupDelay(PT := STARTUP_DELAY);
_CheckSafetyStatus();

// --- Subsystem safety gating ---
IF NOT GVL_Simulation.bActive THEN
    IF _eState <> E_SafetyState.OK THEN
        // Disable heat zones when not safe (PRG_SHARK gates PRG_HEAT_ZONE behind SafetyOk)
        GVL_System.bGlobalSafetyOK := FALSE;
    ELSE
        GVL_System.bGlobalSafetyOK := TRUE;
    END_IF

    // Enable MFCs when voltage comes on
    IF _rtVoltageOn.Q THEN
        _EnableAllMFCs();
        GVL_ErrorLogger.Logger.LogInfo(
            sSource  := 'SafetyManager',
            sContext := 'heater voltage detected - MFCs enabled'
        );
    END_IF

    IF _ftVoltageOff.Q THEN
        GVL_ErrorLogger.Logger.LogInfo(
            sSource  := 'SafetyManager',
            sContext := 'heater voltage OFF'
        );
    END_IF
ELSE
    GVL_System.bGlobalSafetyOK := TRUE;
END_IF

METHOD PUBLIC Init : BOOL
VAR_INPUT
    refFlowSubsystem : REFERENCE TO FB_FlowSubsystem;
END_VAR
    IF NOT __ISVALIDREF(refFlowSubsystem) THEN
        GVL_ErrorLogger.Logger.LogError(
            sSource  := 'SafetyManager.Init',
            eErrorId := E_ErrorId.ERR_GEN_NULL_POINTER,
            sContext := 'invalid flow subsystem reference'
        );
        RETURN;
    END_IF

    _ipFlowSubsystem REF= refFlowSubsystem;
    _fbError.Init('SafetyManager');
    _bInitialized := TRUE;
    Init := TRUE;
END_METHOD

METHOD PRIVATE _CheckSafetyStatus
    // Heartbeat — always signal running
    GVL_Safety.SafetyRunning := TRUE;

    // Detect loss of safe state
    _rtNotSafe(CLK := GVL_Safety.SafetyOk);
    IF _rtNotSafe.Q THEN
        _nInitStep := 0;
        _eState := E_SafetyState.ERROR;
    END_IF

    CASE _eState OF
        E_SafetyState.ERROR:
            // The state machine boots in ERROR while TwinSAFE is still negotiating,
            // so suppress the logged trip on the very first pass — otherwise every
            // startup emits a spurious 'safety error'. A genuine, persistent trip is
            // still surfaced by the gated _fbError.Raise('TwinSAFE not OK') below,
            // which only fires after STARTUP_DELAY.
            _rtError(CLK := _eState = E_SafetyState.ERROR);
            IF _rtError.Q AND NOT _bFirstCycle THEN
                GVL_ErrorLogger.Logger.LogError(
                    sSource  := 'SafetyManager',
                    eErrorId := E_ErrorId.ERR_CTRL_SAFETY_TRIPPED,
                    sContext := 'safety error'
                );
            END_IF
            _eState := E_SafetyState.INIT;
            _bFirstCycle := FALSE;

        E_SafetyState.INIT:
            CASE _nInitStep OF
                0:
                    // Step 1: Assert restart, clear acknowledge
                    GVL_Safety.SafetyErrorAcknowledge := FALSE;
                    GVL_Safety.SafetyRestart := TRUE;
                    IF _tonSafetyStep.Q THEN
                        _nInitStep := 1;
                        _tonSafetyStep.IN := FALSE;
                    END_IF

                1:
                    // Step 2: Assert error acknowledge
                    GVL_Safety.SafetyErrorAcknowledge := TRUE;
                    IF _tonSafetyStep.Q THEN
                        _nInitStep := 2;
                        _tonSafetyStep.IN := FALSE;
                    END_IF

                2:
                    // Step 3: Clear both, check if safe state restored
                    GVL_Safety.SafetyRestart := FALSE;
                    GVL_Safety.SafetyErrorAcknowledge := FALSE;
                    _nInitStep := 0;
                    IF GVL_Safety.SafetyOk THEN
                        _eState := E_SafetyState.OK;
                    END_IF
            END_CASE
            _tonSafetyStep(PT := SAFETY_STEP_TIME);

        E_SafetyState.WAIT_FOR_RESET_BTN:
            IF GVL_Safety.SafetyOk THEN
                _eState := E_SafetyState.OK;
            END_IF

        E_SafetyState.OK:
            IF _tonStartupDelay.Q THEN
                IF NOT GVL_Safety.SafetyOk THEN
                    _eState := E_SafetyState.ERROR;
                END_IF
            END_IF
    END_CASE

    // Simulation override
    IF GVL_Simulation.bActive THEN
        _eState := E_SafetyState.OK;
    END_IF

    // Surface state into the software error plane so subsystem aggregators
    // (FB_TemperatureSubsystem.stFirstError etc.) can see TwinSAFE trips.
    // Only raise after the startup delay elapses — otherwise every boot logs a
    // spurious trip while TwinSAFE is still negotiating.
    IF _eState = E_SafetyState.OK OR GVL_Simulation.bActive THEN
        IF _fbError.IsActive() THEN
            _fbError.Clear();
        END_IF
    ELSIF _tonStartupDelay.Q THEN
        _fbError.Raise(E_ErrorId.ERR_CTRL_SAFETY_TRIPPED, 'TwinSAFE not OK', E_TcEventSeverity.Critical);
    END_IF
END_METHOD

METHOD PRIVATE _CheckVoltage : BOOL
    IF GVL_Simulation.bActive THEN
        _CheckVoltage := TRUE;
        RETURN;
    END_IF
    _CheckVoltage := GVL_Safety.HeaterVoltage > VOLTAGE_THRESHOLD;
END_METHOD

METHOD PRIVATE _EnableAllMFCs
VAR
    i : INT;
    ipController : I_Controller;
END_VAR
    IF NOT __ISVALIDREF(_ipFlowSubsystem) THEN
        GVL_ErrorLogger.Logger.LogError(
            sSource  := 'SafetyManager._EnableAllMFCs',
            eErrorId := E_ErrorId.ERR_GEN_NULL_POINTER,
            sContext := 'flow subsystem reference invalid'
        );
        RETURN;
    END_IF

    FOR i := 1 TO GVL_FlowSystem.FLOW_ZONE_COUNT DO
        ipController := _ipFlowSubsystem.GetControllerByIndex(i);
        IF ipController <> 0 THEN
            ipController.Enable(TRUE);
        END_IF
    END_FOR
END_METHOD

PROPERTY PUBLIC HeaterVoltagePresence : BOOL
    GET
        HeaterVoltagePresence := _bHeaterVoltagePresent;
    END_GET
END_PROPERTY

PROPERTY PUBLIC State : E_SafetyState
    GET
        State := _eState;
    END_GET
END_PROPERTY

PROPERTY PUBLIC IsOk : BOOL
    GET
        IsOk := _eState = E_SafetyState.OK;
    END_GET
END_PROPERTY

// Single source of truth for "is it safe to energize heaters right now".
// Mirrors the gate previously duplicated in PRG_SHARK:
//   IF GVL_Simulation.bActive OR GVL_Safety.SafetyOk THEN PRG_HEAT_ZONE()
// Kept as a pure read (no side effects) so callers can poll safely each cycle.
PROPERTY PUBLIC IsHeatingAllowed : BOOL
    GET
        IsHeatingAllowed := GVL_Simulation.bActive OR GVL_Safety.SafetyOk;
    END_GET
END_PROPERTY

    (* I_Errorable implementation — exposes TwinSAFE state to subsystem error aggregators. *)
METHOD PUBLIC IsError : BOOL
    IsError := _fbError.IsActive();
END_METHOD

METHOD PUBLIC GetError : ST_Error
    GetError := _fbError.GetError();
END_METHOD

END_FUNCTION_BLOCK

(* ---- FB_SignalLightController.st ---- *)
(*
FB_SignalLightController — Drives the three-color signal tower based on machine state.

Owned by PRG_SHARK; initialized once in section 8, called every scan in section 6b.
Signal lights are exclusively controlled by this FB — they are NOT manually settable
via FB_CommandReceiver.

State priority (highest first):
  ERROR  → RED   on, YELLOW off, GREEN off  (bError = TRUE)
  BUSY   → YELLOW on, GREEN  off, RED   off  (bBusy = TRUE, bError = FALSE)
  IDLE   → GREEN  on, YELLOW off, RED   off  (bBusy = FALSE, bError = FALSE)
*)
FUNCTION_BLOCK FB_SignalLightController
VAR
    _ipGreen  : I_DigitalOutput;
    _ipYellow : I_DigitalOutput;
    _ipRed          : I_DigitalOutput;
    _bInitialized   : BOOL := FALSE;
END_VAR

METHOD PUBLIC Init : BOOL
VAR_INPUT
    ipGreen  : I_DigitalOutput;
    ipYellow : I_DigitalOutput;
    ipRed    : I_DigitalOutput;
END_VAR
    IF ipGreen = 0 OR ipYellow = 0 OR ipRed = 0 THEN RETURN; END_IF
    _ipGreen  := ipGreen;
    _ipYellow := ipYellow;
    _ipRed    := ipRed;
    _bInitialized := TRUE;
    Init          := TRUE;
END_METHOD

METHOD PUBLIC Execute
VAR_INPUT
    stStatus : ST_SequenceStatus;
END_VAR
    IF NOT _bInitialized THEN RETURN; END_IF

    IF stStatus.bError THEN
        _ipRed.SetOutput(TRUE);
        _ipYellow.SetOutput(FALSE);
        _ipGreen.SetOutput(FALSE);
    ELSIF stStatus.bBusy THEN
        _ipYellow.SetOutput(TRUE);
        _ipGreen.SetOutput(FALSE);
        _ipRed.SetOutput(FALSE);
    ELSE
        _ipGreen.SetOutput(TRUE);
        _ipYellow.SetOutput(FALSE);
        _ipRed.SetOutput(FALSE);
    END_IF
END_METHOD

END_FUNCTION_BLOCK

(* ---- FB_TelemetryPublisher.st ---- *)
(*
FB_TelemetryPublisher (Shark) — Detailed per-channel telemetry view.

EXTENDS FB_TelemetryPublisherBase (in Lib) which owns the six shared
subsystem refs, Init plumbing, and the per-scan orchestration body. This
derived FB overrides each hook to write into the Shark-specific
ST_MachineTelemetry struct, including the hand-mapped DIOS_ array.

ADS symbol paths:
    READ: PRG_Telemetry.fbTelemetryPublisher.stTelemetry         (ST_MachineTelemetry) — live, updated every scan
    READ: PRG_Telemetry.fbTelemetryPublisher.stSnapshotTelemetry (ST_MachineTelemetry) — frozen at first error; valid when bSnapshotValid = TRUE
    READ: PRG_Telemetry.fbTelemetryPublisher.stSnapshotError     (ST_Error)            — which error triggered the freeze
    READ: PRG_Telemetry.fbTelemetryPublisher.bSnapshotValid      (BOOL)                — FALSE until a snapshot is captured

Snapshot lifecycle:
    Error fires → bSnapshotValid := TRUE, stSnapshotTelemetry frozen, ADSLOG written.
    Snapshot persists through error-clear. Call fbTelemetryPublisher.ResetSnapshot()
    (e.g. from a sequence or command receiver) to re-arm for the next fault.
*)
FUNCTION_BLOCK FB_TelemetryPublisher EXTENDS FB_TelemetryPublisherBase
VAR_OUTPUT
    stTelemetry         : ST_MachineTelemetry;
    // Error-time snapshot fields. Frozen once per unique fault; persist until ResetSnapshot() is called.
    stSnapshotTelemetry : ST_MachineTelemetry; // frozen copy of stTelemetry at error moment
    stSnapshotError     : ST_Error;            // which error triggered the freeze
    bSnapshotValid      : BOOL;                // FALSE at startup; TRUE once a snapshot has been captured
END_VAR

    SUPER^();

METHOD PUBLIC Init : BOOL
VAR_INPUT
    refValveSub    : REFERENCE TO FB_ValveSubsystem;
    refFlowSub     : REFERENCE TO FB_FlowSubsystem;
    refPressureSub : REFERENCE TO FB_PressureSubsystem;
    refTempSub     : REFERENCE TO FB_TemperatureSubsystem;
    refDISub       : REFERENCE TO FB_DigitalInputSubsystem;
    refDOSub       : REFERENCE TO FB_DigitalOutputSubsystem;
END_VAR
    Init := SUPER^.InitSubsystems(
        refValveSub    := refValveSub,
        refFlowSub     := refFlowSub,
        refPressureSub := refPressureSub,
        refTempSub     := refTempSub,
        refDISub       := refDISub,
        refDOSub       := refDOSub);
END_METHOD

METHOD PUBLIC SetCommandIndex
VAR_INPUT
    nCommandIndex : DINT;
END_VAR
    stTelemetry.STAT_[1].CommandIndex := nCommandIndex;
END_METHOD

METHOD PROTECTED _UpdateValves
VAR
    i       : INT;
    ipValve : I_Valve;
END_VAR
    FOR i := 1 TO GVL_ValveSystem.VALVE_COUNT DO
        ipValve := _refValveSub.GetValveByIndex(nValveId := i);
        IF ipValve <> 0 THEN
            stTelemetry.VALV_[i].Open := ipValve.IsOpen();
        END_IF
    END_FOR
END_METHOD

METHOD PROTECTED _UpdateMFC
VAR
    ipSensor     : I_Sensor;
    ipController : I_Controller;
    status       : ST_ControllerStatus;
    i            : INT;
END_VAR
    FOR i := 1 TO GVL_FlowSystem.FLOW_ZONE_COUNT DO
        ipSensor     := _refFlowSub.GetSensorByIndex(nZone := i);
        ipController := _refFlowSub.GetControllerByIndex(nZone := i);
        IF ipSensor <> 0 THEN
            stTelemetry.MFCT_[i].Measure := TO_REAL(ipSensor.GetMeasurement());
        END_IF
        IF ipController <> 0 THEN
            status := ipController.GetStatus();
            stTelemetry.MFCT_[i].SetPoint      := TO_REAL(status.rSetpoint);
            stTelemetry.MFCT_[i].TargetReached := status.bAtSetpoint;
        END_IF
    END_FOR
END_METHOD

METHOD PROTECTED _UpdatePressureSensors
VAR
    ipSensor : I_Sensor;
    i        : INT;
END_VAR
    FOR i := 1 TO GVL_PressureSystem.SENSOR_COUNT DO
        ipSensor := _refPressureSub.GetSensorByIndex(nSensor := i);
        IF ipSensor <> 0 THEN
            stTelemetry.PSNS_[i].Pressure := TO_REAL(ipSensor.GetMeasurement());
        END_IF
    END_FOR
END_METHOD

METHOD PROTECTED _UpdatePressureControllers
VAR
    ipController : I_Controller;
    ipSensor     : I_Sensor;
    status       : ST_ControllerStatus;
    i            : INT;
END_VAR
    FOR i := 1 TO GVL_PressureSystem.CONTROLLER_COUNT DO
        ipController := _refPressureSub.GetControllerByIndex(nCtrl := i);
        IF ipController <> 0 THEN
            status := ipController.GetStatus();
            stTelemetry.PCTR_[i].Enable        := status.bEnabled;
            stTelemetry.PCTR_[i].SetPoint      := TO_REAL(status.rSetpoint);
            stTelemetry.PCTR_[i].ValveOutput   := TO_REAL(status.rOutput);
            stTelemetry.PCTR_[i].TargetReached := status.bAtSetpoint;
        END_IF
        ipSensor := _refPressureSub.GetControllerAsSensorByIndex(nCtrl := i);
        IF ipSensor <> 0 THEN
            stTelemetry.PCTR_[i].Measure := TO_REAL(ipSensor.GetMeasurement());
        END_IF
    END_FOR
END_METHOD

METHOD PROTECTED _UpdateHeaters
VAR
    iZone      : INT;
    c          : INT;
    nCount     : INT;
    nGlobalIdx : INT;
    ipChannel  : I_Controller;
    stCtrl     : ST_ControllerStatus;
END_VAR
    // Detailed (per-CHANNEL) view: one slot per FB_BeckhoffTempController.
    FOR iZone := 1 TO GVL_TemperatureZones.CONTROLLABLE_ZONE_MAX DO
        nCount := GVL_TemperatureZoneConfig.ZONE_CONFIG[iZone].nChannelCount;
        FOR c := 1 TO nCount DO
            nGlobalIdx := _refTempSub.GetChannelGlobalIndex(eZone := iZone, nChannelIdx := c);
            IF nGlobalIdx < 1 THEN CONTINUE; END_IF
            ipChannel := _refTempSub.GetChannel(eZone := iZone, nChannelIdx := c);
            IF ipChannel = 0 THEN CONTINUE; END_IF
            stCtrl := ipChannel.GetStatus();
            stTelemetry.HETR_[nGlobalIdx].Enable             := stCtrl.bEnabled;
            stTelemetry.HETR_[nGlobalIdx].TempAvg            := TO_REAL(stCtrl.rMeasuredValue);
            stTelemetry.HETR_[nGlobalIdx].SP                 := TO_REAL(stCtrl.rSetpoint);
            stTelemetry.HETR_[nGlobalIdx].TemperatureReached := stCtrl.bAtSetpoint;
            stTelemetry.HETR_[nGlobalIdx].Status             := SEL(
                stCtrl.stError.eErrorId = E_ErrorId.NO_ERROR, INT#1, INT#0);
        END_FOR
    END_FOR

    // Per-ZONE summary (zone aggregate from FB_HeatZone).
    _UpdateZoneHeaters(stTelemetry.ZHETR_);
END_METHOD

METHOD PROTECTED _UpdateDigitalIO
    // Camera lights
    stTelemetry.DIOS_[E_DIOIdentifier.LGHT_CMR_SIDE].State :=
        _refDOSub.GetStateByIndex(nOutput := E_DigitalOutputIdentifier.LGHT_CMR_SIDE);
    stTelemetry.DIOS_[E_DIOIdentifier.LGHT_CMR_TOP].State :=
        _refDOSub.GetStateByIndex(nOutput := E_DigitalOutputIdentifier.LGHT_CMR_TOP);

    // Chiller
    stTelemetry.DIOS_[E_DIOIdentifier.CHIL_PWR].State :=
        _refDOSub.GetStateByIndex(nOutput := E_DigitalOutputIdentifier.CHIL_PWR);

    // Signal lights
    stTelemetry.DIOS_[E_DIOIdentifier.LGHT_SGN_RED].State :=
        _refDOSub.GetStateByIndex(nOutput := E_DigitalOutputIdentifier.LGHT_SGN_RED);
    stTelemetry.DIOS_[E_DIOIdentifier.LGHT_SGN_YEL].State :=
        _refDOSub.GetStateByIndex(nOutput := E_DigitalOutputIdentifier.LGHT_SGN_YEL);
    stTelemetry.DIOS_[E_DIOIdentifier.LGHT_SGN_GRN].State :=
        _refDOSub.GetStateByIndex(nOutput := E_DigitalOutputIdentifier.LGHT_SGN_GRN);

    // Door locks
    stTelemetry.DIOS_[E_DIOIdentifier.LOCK_DOOR_FL].State :=
        _refDOSub.GetStateByIndex(nOutput := E_DigitalOutputIdentifier.LOCK_DOOR_FL);
    stTelemetry.DIOS_[E_DIOIdentifier.LOCK_DOOR_FR].State :=
        _refDOSub.GetStateByIndex(nOutput := E_DigitalOutputIdentifier.LOCK_DOOR_FR);

    // Door sensors (9 proximity sensors)
    stTelemetry.DIOS_[E_DIOIdentifier.PRXS_DOOR_LT].State :=
        _refDISub.GetStateByIndex(nInput := E_DigitalInputIdentifier.PRXS_DOOR_LT);
    stTelemetry.DIOS_[E_DIOIdentifier.PRXS_DOOR_LM].State :=
        _refDISub.GetStateByIndex(nInput := E_DigitalInputIdentifier.PRXS_DOOR_LM);
    stTelemetry.DIOS_[E_DIOIdentifier.PRXS_DOOR_LB].State :=
        _refDISub.GetStateByIndex(nInput := E_DigitalInputIdentifier.PRXS_DOOR_LB);
    stTelemetry.DIOS_[E_DIOIdentifier.PRXS_DOOR_RT].State :=
        _refDISub.GetStateByIndex(nInput := E_DigitalInputIdentifier.PRXS_DOOR_RT);
    stTelemetry.DIOS_[E_DIOIdentifier.PRXS_DOOR_RM].State :=
        _refDISub.GetStateByIndex(nInput := E_DigitalInputIdentifier.PRXS_DOOR_RM);
    stTelemetry.DIOS_[E_DIOIdentifier.PRXS_DOOR_RB].State :=
        _refDISub.GetStateByIndex(nInput := E_DigitalInputIdentifier.PRXS_DOOR_RB);
    stTelemetry.DIOS_[E_DIOIdentifier.PRXS_DOOR_BML].State :=
        _refDISub.GetStateByIndex(nInput := E_DigitalInputIdentifier.PRXS_DOOR_BML);
    stTelemetry.DIOS_[E_DIOIdentifier.PRXS_DOOR_BMR].State :=
        _refDISub.GetStateByIndex(nInput := E_DigitalInputIdentifier.PRXS_DOOR_BMR);
    stTelemetry.DIOS_[E_DIOIdentifier.PRXS_DOOR_BMB].State :=
        _refDISub.GetStateByIndex(nInput := E_DigitalInputIdentifier.PRXS_DOOR_BMB);

    // Chuck vacuum pump
    stTelemetry.DIOS_[E_DIOIdentifier.PUMP_CHK_VAC].State :=
        _refDOSub.GetStateByIndex(nOutput := E_DigitalOutputIdentifier.PUMP_CHK_VAC);

    // Chuck valves
    stTelemetry.DIOS_[E_DIOIdentifier.VALV_CHK_LZ1].State :=
        _refDOSub.GetStateByIndex(nOutput := E_DigitalOutputIdentifier.VALV_CHK_LZ1);
    stTelemetry.DIOS_[E_DIOIdentifier.VALV_CHK_LZ2].State :=
        _refDOSub.GetStateByIndex(nOutput := E_DigitalOutputIdentifier.VALV_CHK_LZ2);
    stTelemetry.DIOS_[E_DIOIdentifier.VALV_CHK_LZ3].State :=
        _refDOSub.GetStateByIndex(nOutput := E_DigitalOutputIdentifier.VALV_CHK_LZ3);
    stTelemetry.DIOS_[E_DIOIdentifier.VALV_CHK_VENT].State :=
        _refDOSub.GetStateByIndex(nOutput := E_DigitalOutputIdentifier.VALV_CHK_VENT);

    // 23: HETR_VOLT_ON — DO
    stTelemetry.DIOS_[E_DIOIdentifier.HETR_VOLT_ON].State :=
        _refDISub.GetStateByIndex(nInput := E_DigitalInputIdentifier.HETR_VOLT_ON);

    // Safety — DI
    stTelemetry.DIOS_[E_DIOIdentifier.SAFE_STO_ON].State :=
        _refDISub.GetStateByIndex(nInput := E_DigitalInputIdentifier.SAFE_STO_ON);
    stTelemetry.DIOS_[E_DIOIdentifier.SAFE_OVERRIDE].State := TRUE; // Always TRUE on Shark
END_METHOD

METHOD PROTECTED _UpdateSequenceStateTelemetry
VAR
    stSeqStatus : ST_SequenceStatus;
    ipSensor    : I_Sensor;
END_VAR
    // Read sequence state from PRG_Sequence via GetStatus() method
    stSeqStatus := PRG_Sequence.GetStatus();

    // Convert E_Sequence enum to INT for MachineState
    stTelemetry.STAT_[1].MachineState := stSeqStatus.eActiveSequence;

    // Progress is already a percentage (0-100)
    stTelemetry.STAT_[1].SubState := REAL_TO_INT(stSeqStatus.rProgress);
    stTelemetry.STAT_[1].SubStateCount := 100;

    // Error ID: non-zero if error state
    IF stSeqStatus.bError THEN
        stTelemetry.STAT_[1].ErrorID := UDINT_TO_INT(stSeqStatus.stLastError.eErrorId);
    ELSE
        stTelemetry.STAT_[1].ErrorID := 0;
    END_IF

    // Track last purged bubblers (A-side precursor, B-side reactant)
    stTelemetry.STAT_[1].LastPrecursorIndex := stSeqStatus.nLastPurgedBubblerA;
    stTelemetry.STAT_[1].LastReactantIndex  := stSeqStatus.nLastPurgedBubblerB;

    // A-side temperature (single monitor sensor — no heater)
    ipSensor := PRG_TEMPERATURE_SENSOR.aipMonitorSensors[E_TemperatureMonitorZone.SENS_A_SIDE];
    IF ipSensor <> 0 THEN
        stTelemetry.STAT_[1].TempAside := TO_REAL(ipSensor.GetMeasurement());
    ELSE
        stTelemetry.STAT_[1].TempAside := 0.0;
    END_IF

    // B-side temperature (single monitor sensor — no heater)
    ipSensor := PRG_TEMPERATURE_SENSOR.aipMonitorSensors[E_TemperatureMonitorZone.SENS_B_SIDE];
    IF ipSensor <> 0 THEN
        stTelemetry.STAT_[1].TempBside := TO_REAL(ipSensor.GetMeasurement());
    ELSE
        stTelemetry.STAT_[1].TempBside := 0.0;
    END_IF

    // Chamber temperature/humidity — on Shark the ambient TH sensor serves as the
    // chamber sensor. MACH_[1] is already populated by _UpdateMachineSpecific (called
    // one line earlier in FB_TelemetryPublisherBase), so simply alias it here.
    stTelemetry.STAT_[1].TempChamber := stTelemetry.MACH_[1].AmbTemperature;
    stTelemetry.STAT_[1].HumiChamber := stTelemetry.MACH_[1].AmbHumidity;

    // Sample hold state
    stTelemetry.STAT_[1].isSampleHold := (stSeqStatus.eActiveSequence = E_Sequence.ChuckVacuumHold);

    // Machine firmware version
    stTelemetry.STAT_[1].sVersion := GVL_Version.stLibVersion.sVersion;
END_METHOD

// Freeze stTelemetry into snapshot storage on a new fault edge.
// Called at most once per unique error — not every scan.
METHOD PROTECTED _OnErrorCapture
VAR_INPUT
    stError : ST_Error;
END_VAR
VAR
    sMsg : STRING(255);
END_VAR
    stSnapshotTelemetry := stTelemetry;
    stSnapshotError     := stError;
    bSnapshotValid      := TRUE;

    sMsg := CONCAT('snapshot frozen for ', TO_STRING(stError.eErrorId));
    sMsg := CONCAT(sMsg, CONCAT(' [', CONCAT(stError.sSource, ']')));
    GVL_ErrorLogger.Logger.LogEvent(
        sSource   := 'Shark.TelemetryPublisher',
        eEventId  := E_EventId.EVT_INFO,
        sContext  := sMsg,
        eSeverity := E_TcEventSeverity.Warning
    );
END_METHOD

// Collect Shark machine-specific errors (safety manager) not covered by
// the shared subsystems. Called only when all four shared subsystems report
// no active error.
METHOD PROTECTED _CollectMachineSpecificError : ST_Error
    IF PRG_SHARK.fbSafetyManager.IsError() THEN
        _CollectMachineSpecificError := PRG_SHARK.fbSafetyManager.GetError();
        RETURN;
    END_IF
    _CollectMachineSpecificError.eErrorId := E_ErrorId.NO_ERROR;
END_METHOD

// Clear bSnapshotValid on operator reset.
// stSnapshotTelemetry is intentionally preserved — it remains readable as
// a historical record; bSnapshotValid = FALSE signals it is stale.
METHOD PROTECTED _OnSnapshotReset
    bSnapshotValid := FALSE;
END_METHOD

// Write ambient temperature and humidity into MACH_[1].
// Temperature is read from PRG_TEMPERATURE_SENSOR (SENS_CHAMBER — the TH sensor temperature channel).
// Humidity is read from PRG_HUMIDITY_SENSOR (AMBT_HUMID — the TH sensor humidity channel).
// Called once per scan by FB_TelemetryPublisherBase via the _UpdateMachineSpecific hook.
METHOD PROTECTED _UpdateMachineSpecific
VAR
    ipSensor : I_Sensor;
END_VAR
    // Ambient temperature (TH sensor — temperature channel, wired as SENS_CHAMBER)
    ipSensor := PRG_TEMPERATURE_SENSOR.aipMonitorSensors[E_TemperatureMonitorZone.SENS_CHAMBER];
    IF ipSensor <> 0 THEN
        stTelemetry.MACH_[1].AmbTemperature := TO_REAL(ipSensor.GetMeasurement());
    ELSE
        stTelemetry.MACH_[1].AmbTemperature := 0.0;
    END_IF

    // Ambient humidity (TH sensor — humidity channel)
    ipSensor := PRG_HUMIDITY_SENSOR.ipSensor;
    IF ipSensor <> 0 THEN
        stTelemetry.MACH_[1].AmbHumidity := TO_REAL(ipSensor.GetMeasurement());
    ELSE
        stTelemetry.MACH_[1].AmbHumidity := 0.0;
    END_IF
END_METHOD
